// TwinCAT 3 PLC project System
// ProgramVersion: 3.1.4023.0
// libraries:
//   Tc2_MC2, * (Beckhoff Automation GmbH)
//   Tc2_MC2_Drive, * (Beckhoff Automation GmbH)
//   Tc2_Standard, * (Beckhoff Automation GmbH)
//   Tc2_System, * (Beckhoff Automation GmbH)
//   Tc3_Module, * (Beckhoff Automation GmbH)
// project tree:
//   00_Internal PackAL/DUTs/ E_PMLState.TcDUT (not stored), E_PMLUnitMode.TcDUT
//   00_Internal PackAL/POUs/ PS_PackML_StateMachine_Auto.TcPOU, PS_PackML_StateMachine_Maintenance.TcPOU, PS_PackML_StateMachine_Manual.TcPOU, PS_PackML_StateMachine_SemiAuto.TcPOU, PS_UnitModeManager.TcPOU
//   01_Submodules/ FB_Axis.TcPOU, FB_MPG.TcPOU
//   02_Subsystems/ FB_Stage.TcPOU
//   03_Machine/ FB_Machine.TcPOU
//   04_Application/ MAIN.TcPOU
//   05_Visu/ FB_Visu.TcPOU, HMI.TcVIS, TAB_Simulation.TcVIS
//   DUTs/ ST_MC_Base.TcDUT, ST_MC_CMD.TcDUT, ST_MC_Reset.TcDUT, ST_MC_Status.TcDUT
//   / GlobalTextList.TcGTLO, PlcTask.TcTTO, Visualization Manager.TcVMO (not stored), VISU_TASK.TcTTO
//   GVLs/ GVL_SA.TcGVL, Temp.TcGVL
//   POUs/ FB_MotorControl.TcPOU, ModbusTCP_Test.TcPOU
// real-time tasks:
//   TASK PlcTask: cycle T#10ms, priority 20, ADS port 350
//   TASK VISU_TASK: cycle T#100000us, priority 30, ADS port 351
// motion (NC):
//   TASK NC-Task 1 SAF: cycle T#2ms, priority 4, ADS port 501
//   TASK NC-Task 1 SVB: cycle T#10ms, priority 8, ADS port 511
//   AXIS Axis 2 (id 2)
//     OtherSettings: AllowMotionCmdToSlave=true
//     encoder EncType=19
//       EncPara: MaxCount=#xffffffff
//     drive DrvType=16
//       DrvPara: MaxCount=#xffffffff, DriveControlDWord=#x00020000
//         Analog: TorqueSetpointScale=10, ScaleFactorActTorque=0.1
//         TimeComp: TaskDelayCycles=1
//     controller CtrType=1
//       CtrPara: PriorControlFactor=1
//         Observer: BandWidth=20
// I/O:
//   DEVICE Device 3 (EtherCAT), AmsNetId 129.169.49.186.4.1
//     Term 1 (EK1100) [EK1100 EtherCAT Coupler (2A E-Bus)] (disabled)
//       Term 2 (EL1114)
//       Term 3 (EL1809) [EL1809 16Ch. Dig. Input 24V, 3ms]
//       Term 4 (EL1809) [EL1809 16Ch. Dig. Input 24V, 3ms]
//       Term 5 (EL2008) [EL2008 8Ch. Dig. Output 24V, 0.5A]
//       Term 6 (EL2809) [EL2809 16Ch. Dig. Output 24V, 0.5A]
//       Term 7 (EL3068) [EL3068 8Ch. Ana. Input 0-10V]
//       Term 8 (EL3058) [EL3058 8Ch. Ana. Input 4-20mA]
//       Term 9 (EL4002) [EL4002 2Ch. Ana. Output 0-10V, 12bit]
//       Term 10 (EL5101) [EL5101 1Ch. Inc. Encoder 5V]
//       Term 11 (EK1110) [EK1110 EtherCAT extension]
//   DEVICE Device 1 (EtherCAT) (disabled), AmsNetId 192.168.1.163.2.1
//     Term 1 (EK1200) [EK1200-5000 EtherCAT Power supply (2A E-Bus)]
//       Term 13 (EL1114) [EL1114 4Ch. Dig. Input 24V, 10µs, Sensor Power]
//       Term 14 (EL1809) [EL1809 16Ch. Dig. Input 24V, 3ms]
//       Term 15 (EL1809) [EL1809 16Ch. Dig. Input 24V, 3ms]
//       Term 16 (EL2008) [EL2008 8Ch. Dig. Output 24V, 0.5A]
//       Term 17 (EL2809) [EL2809 16Ch. Dig. Output 24V, 0.5A]
//       Term 18 (EL3068) [EL3068 8Ch. Ana. Input 0-10V]
//       Term 19 (EL3058) [EL3058 8Ch. Ana. Input 4-20mA]
//       Term 20 (EL4002) [EL4002 2Ch. Ana. Output 0-10V, 12bit]
//       Term 21 (EL5101) [EL5101 1Ch. Inc. Encoder 5V]
//       Term 22 (EK1110) [EK1110 EtherCAT extension]
//   DEVICE Device 5 (NOV-DP-RAM)
// variable links:
//   System Instance <-> Device 3 (EtherCAT)/Term 1 (EK1100)/Term 10 (EL5101)
//     PlcTask Inputs/MAIN.fbMachine.fbMPG.EncoderValue <-> ENC Status compact/Counter value
//   System Instance <-> NC-Task 1 SAF/Axes/Axis 2
//     PlcTask Inputs/GVL_SA.Motor1.AxisRef.NcToPlc <-> Outputs/ToPlc
//     PlcTask Outputs/GVL_SA.Motor1.AxisRef.PlcToNc <-> Inputs/FromPlc

CONFIGURATION System
    RESOURCE PLC ON TwinCAT3
        TASK PlcTask(INTERVAL := T#10ms, PRIORITY := 20);
        TASK VISU_TASK(INTERVAL := T#100000us, PRIORITY := 30);
        PROGRAM MAIN WITH PlcTask : MAIN;
        PROGRAM VisuElems_Visu_Prg WITH VISU_TASK : VisuElems.Visu_Prg;
    END_RESOURCE
END_CONFIGURATION

// ---- 00_Internal PackAL/DUTs/E_PMLUnitMode.TcDUT
{attribute 'qualified_only'}
{attribute 'strict'}
TYPE E_PMLUnitMode :
(
	UNDEFINED		:=  0,
	AUTOMATIC		:=  1,
	MAINTENANCE 	:=  2,
	MANUAL 			:=  3,
	SEMIAUTOMATIC	:=  4,
	DRYRUN			:=  5,
	USERMODE1		:=  6,
	USERMODE2		:=  7,
	IDLE 			:=  8,
	ESTOP 			:=  9
);
END_TYPE

// ---- DUTs/ST_MC_Base.TcDUT
TYPE ST_MC_Base :
STRUCT
	Busy		:	BOOL;
	Error		:	BOOL;
	ErrrorID	:	UDINT;
END_STRUCT
END_TYPE

// ---- DUTs/ST_MC_CMD.TcDUT
TYPE ST_MC_CMD :
STRUCT
	bExe			: BOOL	;
	lrVelocity		: LREAL	;
	lrAcceleration 	: LREAL ;
	lrDeceleration 	: LREAL ;
	lrJerk 			: LREAL ;
	lrDistance 		: LREAL ; 
	lrPosition 		: LREAL ; 
	EnuDirection 	: MC_Direction ;
	EnuBufferMode 	: MC_BufferMode ; 
	EnuOptions 		: ST_MoveOptions ;
END_STRUCT
END_TYPE

// ---- DUTs/ST_MC_Reset.TcDUT
TYPE ST_MC_Reset:
STRUCT
	
	CMD_Execute	: 	BOOL;
	
	Done		: 	BOOL;
	Busy		:	BOOL;
	Error		:	BOOL;
	ErrrorID	:	UDINT;	

END_STRUCT
END_TYPE

// ---- DUTs/ST_MC_Status.TcDUT
TYPE ST_MC_Status :
STRUCT
	
	Status		:	BOOL;
	Done		:	BOOL;
	Busy		:	BOOL;
	Error		:	BOOL;
	Active		:	BOOL;
	CmdAborted	:	BOOL;
	InVelocity	:	BOOL;
	ErrrorID	:	UDINT;
	
	Value		: 	LREAL;
	Valid		: 	BOOL;
	

END_STRUCT
END_TYPE

// ---- GVLs/GVL_SA.TcGVL
{attribute 'qualified_only'}
VAR_GLOBAL
	Motor1 : FB_MotorControl;	
END_VAR

// ---- GVLs/Temp.TcGVL
{attribute 'qualified_only'}
VAR_GLOBAL
	//GVL_MPG_Value : UINT;
	
	bSwitch1:	BOOL;
	bLED1: BOOL;
	
	
END_VAR

// ---- 04_Application/MAIN.TcPOU
PROGRAM MAIN
VAR
	fbMachine : FB_Machine;	

	Dummy : BOOL := FALSE;
	bTest: BOOL := FALSE;
	
	MAIN_UINT : UINT;
	
END_VAR

// =========================================================

fbMachine();

// =========================================================


//GVL_SA.Motor1.UpdateAll();
GVL_SA.Motor1();

GVL_SA.Motor1.bStateEnable := TRUE;

{IF defined (Pyrometer_Motor)}
	bTest := TRUE;
{END_IF}

Dummy	:= TRUE;

Temp.bLED1 := Temp.bSwitch1;

END_PROGRAM

// ---- 03_Machine/FB_Machine.TcPOU
FUNCTION_BLOCK FB_Machine
VAR_INPUT
	
END_VAR
VAR_OUTPUT
END_VAR
VAR
	// =============== Common variables =========================================================
	bInit								: BOOL;									// True if module parameters are initialized	

		
	
	// =============== Machine elements =========================================================
	// This can be either Submodules or SubSystems
	fbMPG 			: 		FB_MPG ;		//MPG unit
	
	
	
	fbVisu : FB_Visu;
	
		fbGetCurTaskIndex : GETCURTASKINDEX;
	
	// =============== Testing ==================================================================
	_UINT : UINT;
END_VAR

// =========================================================
// Call of actions

//Check for start cycle
//Move to main later.....
//fbGetCurTaskIndex();
//IF _TaskInfo[fbGetCurTaskIndex.index].FirstCycle THEN
//    // The code that you want to be executed at the first cycle
//	eMPGState := INIT_START;
//END_IF


	// Init
	General_Init();

	// Mode and state requests
	//General_Requests();
	
	// Enable for power supply, compressed air control and buttons
	//General_Enable();
	
	// Input variables of separating and sorting modules
	//General_ModuleInputs();
	
	// Output variables
	//General_SetOutput();
	
	// State machine
	//General_StateMachine();
	
	// Visualization
	//General_Visu();
	fbVisu();
	

// =========================================================
//TESTING


	_UINT := fbMPG.Value;

METHOD PRIVATE General_Init
VAR_INPUT
		
END_VAR
// =========================================================
IF NOT bInit THEN
		fbMPG.Start(1234);
		
	// Init done
		bInit := TRUE;
END_IF
// =========================================================
END_METHOD

METHOD PRIVATE Operating_Automatic
VAR_INPUT
END_VAR
END_METHOD

METHOD PRIVATE Operating_Manual
VAR_INPUT
END_VAR
END_METHOD

END_FUNCTION_BLOCK

// ---- 01_Submodules/FB_MPG.TcPOU
FUNCTION_BLOCK FB_MPG
VAR_INPUT
END_VAR
VAR_OUTPUT
END_VAR
VAR
	//Hardware declared here as only one will ever be connected 
	EncoderValue 		AT %I* : UINT;	//Measured Value from Encoder
	SetValueZero	 	AT %Q* : BOOL;	//Request encoder be reset to zero 	
	bX1					AT %I* : BOOL;	//Multipliers
	bX10				AT %I* : BOOL;
	bX100				AT %I* : BOOL;
	bEnabled			AT %I* : BOOL;
	
	
	eMPGState : (INIT_START, WAIT_START, RUNNING, STOPPED);	//MPG state machine defenitions
	
	nMotorStartPoisition	: UINT	;	//Where was the motor at the beginning
	nDeltaPosition			: DINT	;	//Calculated position request change from start
										//Motor value 	nMotorStartPoisition + nDeltaPosition

	nLastEncoderValue		: UINT	;	//Encoder value on last scan cycle
	nDeltaEncoder_PerScan	: DINT	;	//Encoder change per scan
	
END_VAR

CASE eMPGState OF
	INIT_START:												//Holding state
		eMPGState := WAIT_START;
	
	WAIT_START:												//Holding state
		eMPGState := RUNNING;

	RUNNING:
		IF (Error_Scaler OR Error_AxisSelect) THEN			//If current error state
			//nDeltaPosition := 0;							//No change in position possible	
		ELSE
			//Update values
			nDeltaEncoder_PerScan  := nLastEncoderValue - EncoderValue;
			nDeltaPosition := nDeltaPosition + nDeltaEncoder_PerScan * ScaleFactor;			
		END_IF

	STOPPED:
		//Do nothing
END_CASE

nLastEncoderValue := EncoderValue;	//Ensure next scan always sees change in encoder position

PROPERTY PUBLIC Error : Bool
GET
//System in any error or any condition other than running.

Error := FALSE;

IF (Error_AxisSelect OR Error_Scaler) THEN
	Error := TRUE;
END_IF

IF eMPGState <> RUNNING THEN
	Error := TRUE;
END_IF
END_GET
END_PROPERTY

PROPERTY PRIVATE Error_AxisSelect : Bool
GET
END_GET
END_PROPERTY

PROPERTY PRIVATE Error_Scaler : Bool
GET
//Error conditions
IF bX1 AND bX10 THEN
	Error_Scaler := TRUE;
	RETURN;
END_IF

IF bX1 AND bX100 THEN
	Error_Scaler := TRUE;
	RETURN;
END_IF

IF bX10 AND bX100 THEN
	Error_Scaler := TRUE;
	RETURN;
END_IF

IF NOT bX1 AND NOT bX10 AND NOT bX100 THEN
	Error_Scaler := TRUE;
	RETURN;
END_IF

Error_Scaler := FALSE;
END_GET
END_PROPERTY

//Returns the scale factor to be used on the new data
PROPERTY PRIVATE ScaleFactor : UINT
GET
//Depending on what IO is connected send back 1, 10, 100 or set error!
IF bX1 THEN
	ScaleFactor := 1;
END_IF

IF bX10 THEN
	ScaleFactor := 10;
END_IF

IF bX100 THEN
	ScaleFactor := 100;
END_IF
END_GET
END_PROPERTY

METHOD PUBLIC Start
VAR_INPUT
	nMotorStartPoisition	:	UINT ;	//Check that this is passed to the "main"
										//May need to be implicitly defined.
END_VAR
eMPGState := INIT_START;
END_METHOD

PROPERTY Starting : Bool
GET
IF (eMPGState = INIT_START OR eMPGState = WAIT_START) THEN
	Starting := TRUE;
	ELSE
	Starting := FALSE;				
END_IF
END_GET
END_PROPERTY

METHOD PUBLIC Stop
VAR_INPUT
END_VAR
eMPGState := E_PMLState.STOPPED;
END_METHOD

PROPERTY Value : UINT		//Calculated ABS position value requested by MPG, check Error before use.
GET
Value := DINT_TO_UINT(nMotorStartPoisition + nDeltaPosition);
//What is the form needed for motor position??
END_GET
END_PROPERTY

END_FUNCTION_BLOCK

// ---- 05_Visu/FB_Visu.TcPOU
FUNCTION_BLOCK FB_Visu
VAR_INPUT
	nMPGCounter : DINT;
END_VAR
VAR_OUTPUT
END_VAR
VAR
	sDisplayText_MPG : STRING(15);
END_VAR

sDisplayText_MPG := 'Sent';

END_FUNCTION_BLOCK

// ---- POUs/FB_MotorControl.TcPOU
FUNCTION_BLOCK FB_MotorControl
VAR_INPUT
	AxisRef 	:	AXIS_REF;
	//Position
	//Ready
	//Reset
	
END_VAR
VAR_OUTPUT
		error	: BOOL;
END_VAR

(*Internals*)
VAR
	(* Properties *)
	Enabled : BOOL := FALSE;	


	eInitMotor : (START, IN_PROCESS, DONE, ERROR);	
	eMoveABS : (START, IN_PROCESS, DONE, ERROR);

	//stMC_Reset : ST_MC_Reset;
	

	stSA_Reset	:   ST_MC_Status;
	
	
	
	fbMcPower	:	MC_POWER;
	fbMcHome	: 	MC_HOME;
	fbMcJog		:	MC_JOG;
	
	// Global
	bError 		: BOOL	; // := TRUE;
	nErrorID 	: LINT	; //Check type
	
	//Reset
	fbMcReset	:	MC_RESET;
	fbTriggerReset : R_TRIG;
	bResetDone : BOOL := FALSE;
	
	
	
	fbMoveVelocity	: MC_MoveVelocity;
	fbMoveRelative	: MC_MoveRelative;
	fbMoveAbsolute	: MC_MoveAbsolute;
	
	fbHalt	: MC_Halt;
	fbStop	: MC_Stop;
	
	fbSA_GetPosition : MC_ReadActualPosition;
	
	//Input: Command
	bCmdResetExe			:	BOOL	;
	bCmdPowerEnable			:	BOOL	;
	bCmdPowerEnablePositive	:	BOOL	;
	bCmdPowerEnableNegative	:	BOOL	;
	bCmdHomeExecute			:	BOOL	;
	bSA_HomeCamInput	:	BOOL	;
	
	bSA_JogFwd			:	BOOL	;
	bSA_JogRev			:	BOOL	;
	
	bSA_HaltExe			: 	BOOL	;
	bSA_StopExe			: 	BOOL	;
	
	//stStatusMoveVelocity	: ST_MC_CMD	;
	stSA_VelCmd1	: ST_MC_CMD;
	stSA_RelCmd1			: ST_MC_CMD	;
	stSA_AbsCmd1			: ST_MC_CMD	;
	
	//Variables / Parameters
	lrSA_PowerOverride	: LREAL;
	lrSA_HomePosition	: LREAL;
	lrSA_SetPosition	: LREAL;
	lrSA_JogVelocity	: LREAL;
	
	//Status
	//stSA_Reset			: ST_MC_Status;
	stSA_Power			: ST_MC_Status;
	stSA_Home			: ST_MC_Status;
	stSA_SetPosition	: ST_MC_Status;
	stSA_Jog			: ST_MC_Status;
	stSA_GetPosition	: ST_MC_Status;
	
	
	stSA_VelSts1		: ST_MC_Status;
	stSA_MoveRelative		: ST_MC_Status;
	stSA_AbsSts1		: ST_MC_Status;
	
	stSA_Halt			: ST_MC_Status;
	stSA_Stop			: ST_MC_Status;

END_VAR

AxisRef.ReadStatus();
GetStatus();
//Here the state machine needs to be processed or farmed out.



//For a move

//Has position changed from the current target.....






//This should be removed as seperate methods are added.
ExecuteCommands();

PROPERTY bStateEnable : BOOL
GET
bStateEnable := Enabled ;
END_GET
SET
Enabled := bStateEnable;
END_SET
END_PROPERTY

METHOD PRIVATE Enable : BOOL
VAR_INPUT
END_VAR
END_METHOD

METHOD PRIVATE ExecuteCommands : BOOL
VAR_INPUT
END_VAR

VAR
END_VAR
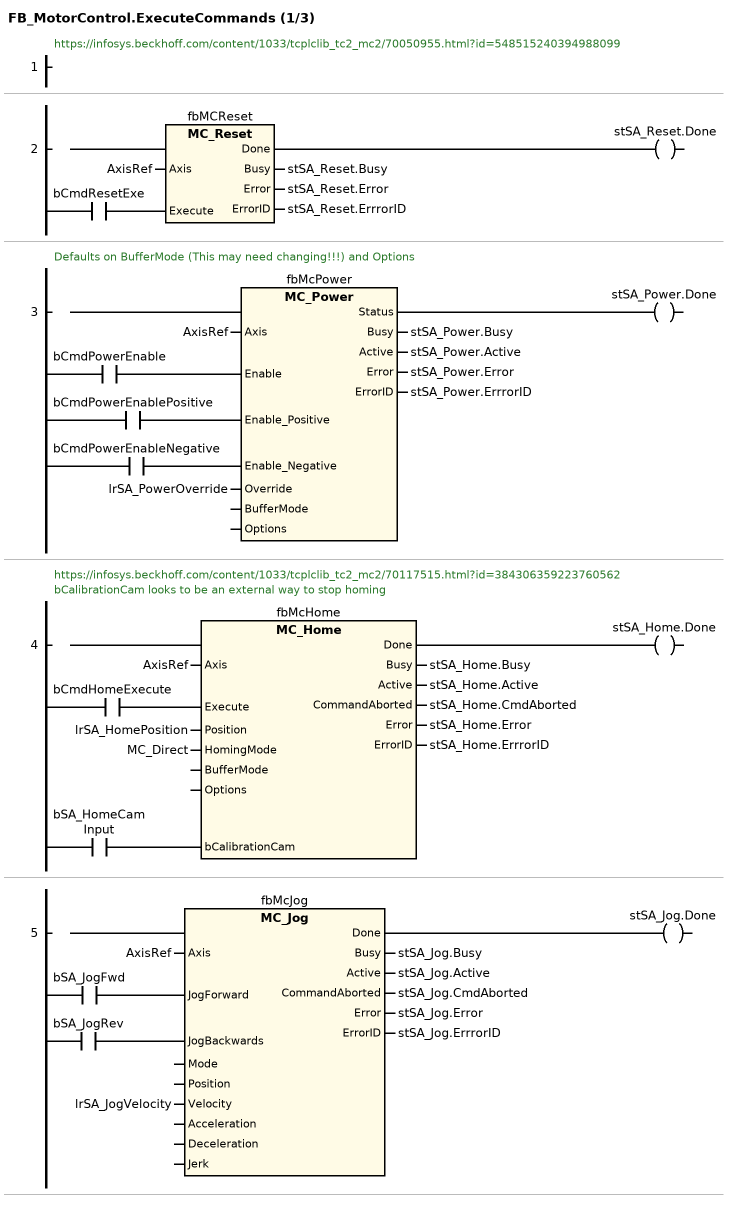
// NETWORK 1
// https://infosys.beckhoff.com/content/1033/tcplclib_tc2_mc2/70050955.html?id=548515240394988099

// NETWORK 2
fbMCReset(
    Axis := AxisRef,
    Execute := bCmdResetExe,
    Busy => stSA_Reset.Busy,
    Error => stSA_Reset.Error,
    ErrorID => stSA_Reset.ErrrorID); // MC_Reset
stSA_Reset.Done := fbMCReset.Done;

// NETWORK 3
// Defaults on BufferMode (This may need changing!!!) and Options
fbMcPower(
    Axis := AxisRef,
    Enable := bCmdPowerEnable,
    Enable_Positive := bCmdPowerEnablePositive,
    Enable_Negative := bCmdPowerEnableNegative,
    Override := lrSA_PowerOverride,
    Busy => stSA_Power.Busy,
    Active => stSA_Power.Active,
    Error => stSA_Power.Error,
    ErrorID => stSA_Power.ErrrorID); // MC_Power
stSA_Power.Done := fbMcPower.Status;

// NETWORK 4
// https://infosys.beckhoff.com/content/1033/tcplclib_tc2_mc2/70117515.html?id=384306359223760562
// bCalibrationCam looks to be an external way to stop homing
fbMcHome(
    Axis := AxisRef,
    Execute := bCmdHomeExecute,
    Position := lrSA_HomePosition,
    HomingMode := MC_Direct,
    bCalibrationCam := bSA_HomeCamInput,
    Busy => stSA_Home.Busy,
    Active => stSA_Home.Active,
    CommandAborted => stSA_Home.CmdAborted,
    Error => stSA_Home.Error,
    ErrorID => stSA_Home.ErrrorID); // MC_Home
stSA_Home.Done := fbMcHome.Done;

// NETWORK 5
fbMcJog(
    Axis := AxisRef,
    JogForward := bSA_JogFwd,
    JogBackwards := bSA_JogRev,
    Velocity := lrSA_JogVelocity,
    Busy => stSA_Jog.Busy,
    Active => stSA_Jog.Active,
    CommandAborted => stSA_Jog.CmdAborted,
    Error => stSA_Jog.Error,
    ErrorID => stSA_Jog.ErrrorID); // MC_Jog
stSA_Jog.Done := fbMcJog.Done;

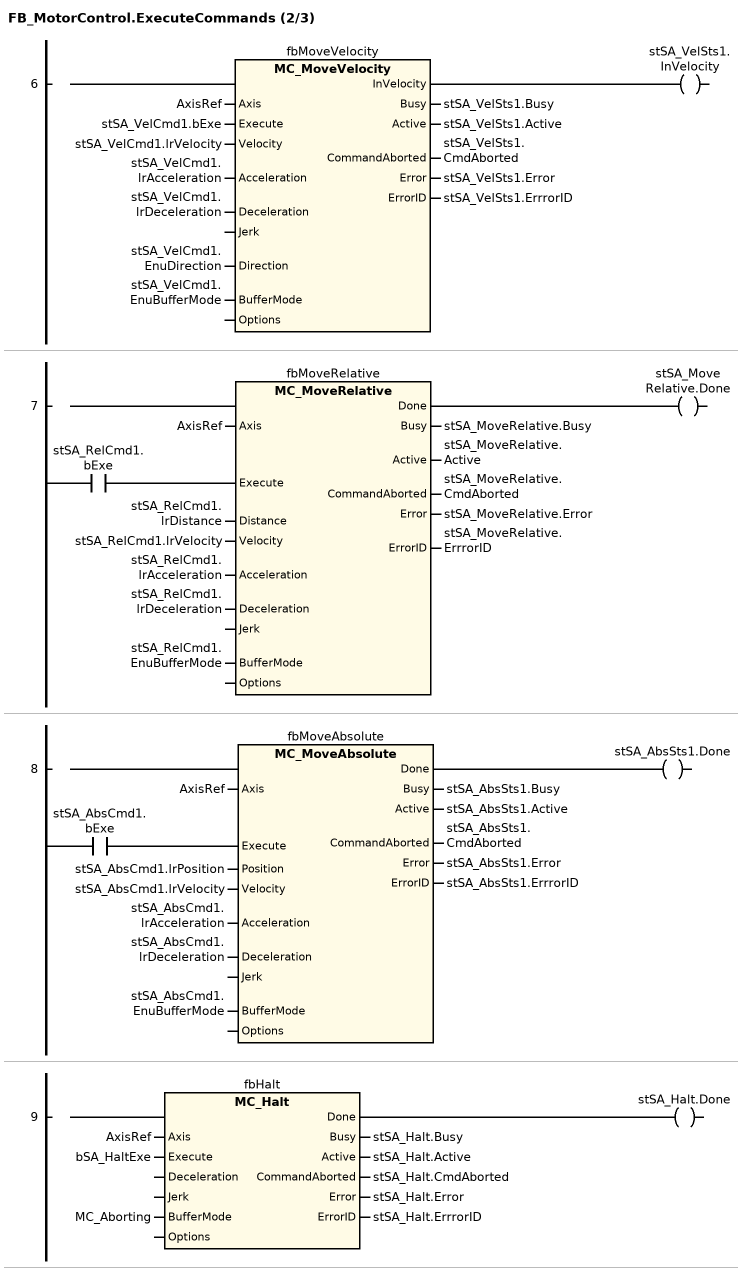
// NETWORK 6
fbMoveVelocity(
    Axis := AxisRef,
    Execute := stSA_VelCmd1.bExe,
    Velocity := stSA_VelCmd1.lrVelocity,
    Acceleration := stSA_VelCmd1.lrAcceleration,
    Deceleration := stSA_VelCmd1.lrDeceleration,
    Direction := stSA_VelCmd1.EnuDirection,
    BufferMode := stSA_VelCmd1.EnuBufferMode,
    Busy => stSA_VelSts1.Busy,
    Active => stSA_VelSts1.Active,
    CommandAborted => stSA_VelSts1.CmdAborted,
    Error => stSA_VelSts1.Error,
    ErrorID => stSA_VelSts1.ErrrorID); // MC_MoveVelocity
stSA_VelSts1.InVelocity := fbMoveVelocity.InVelocity;

// NETWORK 7
fbMoveRelative(
    Axis := AxisRef,
    Execute := stSA_RelCmd1.bExe,
    Distance := stSA_RelCmd1.lrDistance,
    Velocity := stSA_RelCmd1.lrVelocity,
    Acceleration := stSA_RelCmd1.lrAcceleration,
    Deceleration := stSA_RelCmd1.lrDeceleration,
    BufferMode := stSA_RelCmd1.EnuBufferMode,
    Busy => stSA_MoveRelative.Busy,
    Active => stSA_MoveRelative.Active,
    CommandAborted => stSA_MoveRelative.CmdAborted,
    Error => stSA_MoveRelative.Error,
    ErrorID => stSA_MoveRelative.ErrrorID); // MC_MoveRelative
stSA_MoveRelative.Done := fbMoveRelative.Done;

// NETWORK 8
fbMoveAbsolute(
    Axis := AxisRef,
    Execute := stSA_AbsCmd1.bExe,
    Position := stSA_AbsCmd1.lrPosition,
    Velocity := stSA_AbsCmd1.lrVelocity,
    Acceleration := stSA_AbsCmd1.lrAcceleration,
    Deceleration := stSA_AbsCmd1.lrDeceleration,
    BufferMode := stSA_AbsCmd1.EnuBufferMode,
    Busy => stSA_AbsSts1.Busy,
    Active => stSA_AbsSts1.Active,
    CommandAborted => stSA_AbsSts1.CmdAborted,
    Error => stSA_AbsSts1.Error,
    ErrorID => stSA_AbsSts1.ErrrorID); // MC_MoveAbsolute
stSA_AbsSts1.Done := fbMoveAbsolute.Done;

// NETWORK 9
fbHalt(
    Axis := AxisRef,
    Execute := bSA_HaltExe,
    BufferMode := MC_Aborting,
    Busy => stSA_Halt.Busy,
    Active => stSA_Halt.Active,
    CommandAborted => stSA_Halt.CmdAborted,
    Error => stSA_Halt.Error,
    ErrorID => stSA_Halt.ErrrorID); // MC_Halt
stSA_Halt.Done := fbHalt.Done;

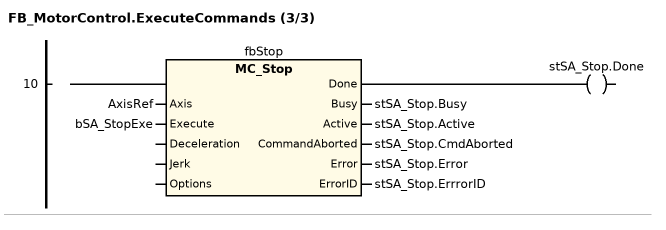
// NETWORK 10
fbStop(
    Axis := AxisRef,
    Execute := bSA_StopExe,
    Busy => stSA_Stop.Busy,
    Active => stSA_Stop.Active,
    CommandAborted => stSA_Stop.CmdAborted,
    Error => stSA_Stop.Error,
    ErrorID => stSA_Stop.ErrrorID); // MC_Stop
stSA_Stop.Done := fbStop.Done;
END_METHOD

METHOD PRIVATE GetStatus : BOOL
VAR_INPUT
END_VAR
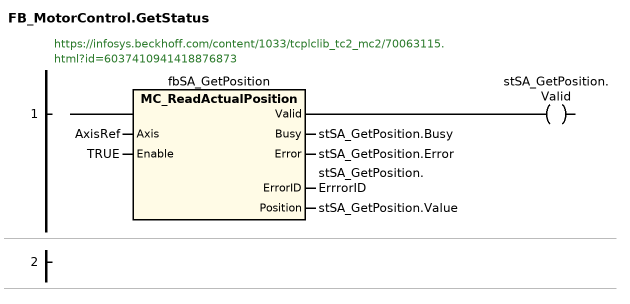
// NETWORK 1
// https://infosys.beckhoff.com/content/1033/tcplclib_tc2_mc2/70063115.html?id=6037410941418876873
fbSA_GetPosition(
    Axis := AxisRef,
    Enable := TRUE,
    Busy => stSA_GetPosition.Busy,
    Error => stSA_GetPosition.Error,
    ErrorID => stSA_GetPosition.ErrrorID,
    Position => stSA_GetPosition.Value); // MC_ReadActualPosition
stSA_GetPosition.Valid := fbSA_GetPosition.Valid;

// NETWORK 2
END_METHOD

METHOD Halt : BOOL
VAR_INPUT
END_VAR
END_METHOD

METHOD PUBLIC MoveAbs : BOOL
VAR_INPUT
	Distance 		: LREAL;
	Velocity 		: LREAL;

//https://infosys.beckhoff.com/content/1033/tcplclib_tc2_mc2/70147595.html?id=4401319670753010232
	mcBufferMode	: MC_BufferMode;
(*  MC_Aborting,			Cancels P1 and  moves to P2
    MC_Buffered,			Moves to P1, stops and moves to P2
    MC_BlendingLow, MC_BlendingPrevious, MC_BlendingNext, MC_BlendingHigh	Change the way speed is blended  BlendingLow would generaly be the one I'd choose. *)
	
END_VAR
VAR
	

END_VAR
(*  It is not needed to wait for the end of a move, will be qued - but do need to ensure Execute operates with a rising edge.
	Not concerned about "loosing" commands, no buffer needed, only the last command matters.*)   

(*
If in Error state ignore.

If "Busy"	Execute == FALSE;

if Execute == FALSE can send new command

*)	

	
	
//CASE fbMoveAbsolute.Execute OF
//	TRUE: 
	
//	IN_PROCESS:

//	DONE:
	
	
//END_CASE

//Does this have meaning.....
MoveAbs := TRUE;
END_METHOD

METHOD Reset : BOOL
VAR_INPUT
	bDriveReset : Bool;
END_VAR
// Indicate that the Reset is in progress
IF NOT bDriveReset THEN
	bResetDone := FALSE;
END_IF

// Trigger
fbTriggerReset(CLK := bDriveReset);

IF fbTriggerReset.Q THEN
	//Is this meant to be sending a halt to the motor at the same time....?
	//If so why not as a command - seems more of a status....
	
	//bHaltDone := FALSE;
	fbMcReset(Execute := TRUE, Axis := AxisRef);
ELSE				
	fbMcReset(Axis := AxisRef); //What happens to the unchanged values - defaults......TEST?
END_IF;
 
// Done / Error 
IF fbMcReset.Done OR fbMcReset.Error THEN
	bError := fbMcReset.Error;
	nErrorID := fbMcReset.ErrorID;
	bResetDone := fbMcReset.Done;
	
	fbMcReset(Execute := FALSE, Axis := AxisRef);
END_IF
END_METHOD

METHOD Stop : BOOL
VAR_INPUT
END_VAR
END_METHOD

END_FUNCTION_BLOCK

// ---- 00_Internal PackAL/POUs/PS_PackML_StateMachine_Auto.TcPOU
FUNCTION_BLOCK PS_PackML_StateMachine_Auto
VAR_INPUT
	Start				: BOOL;
	Hold				: BOOL;
	UnHold				: BOOL;
	Suspend				: BOOL;
	UnSuspend			: BOOL;
	Abort				: BOOL;
	Stop				: BOOL;
	Complete			: BOOL;
	Clear				: BOOL;
	Reset				: BOOL;
	StateComplete		: BOOL;
END_VAR
VAR_OUTPUT
	Status				: WORD;

	ST_Starting			: BOOL;
	ST_Completing		: BOOL;
	ST_Resetting		: BOOL;
	ST_Holding			: BOOL;
	ST_UnHolding		: BOOL;
	ST_Suspending		: BOOL;
	ST_UnSuspending		: BOOL;
	ST_Clearing			: BOOL;
	ST_Stopping			: BOOL;
	ST_Aborting			: BOOL;

	(* State Complete*)
	ST_Execute			: BOOL;
	ST_Complete			: BOOL;
	ST_Idle				: BOOL;
	ST_Held				: BOOL;
	ST_Suspended		: BOOL;
	ST_Stopped			: BOOL;
	ST_Aborted			: BOOL;

	(* additional *)
	Error				: BOOL;
	ErrorID				: DWORD;
	ePMLState			: E_PMLState := E_PMLState.IDLE;
END_VAR
VAR
	ePMLStatePrev		: E_PMLState;
	bStateChange		: BOOL;
	StateCompletePrev	: BOOL;
END_VAR

(* check for state change *)
IF ePMLStatePrev <> ePMLState THEN
	ePMLStatePrev 	:= ePMLState;
	bStateChange	:= TRUE;
ELSE
	bStateChange	:= FALSE;
END_IF


(* change to new state if requested *)
CASE ePMLState OF
	E_PMLState.UNDEFINED:
				(* undefined state *)
				IF bStateChange THEN
					(* transient state *)
					ST_Starting		:= FALSE;
					ST_Completing	:= FALSE;
					ST_Resetting	:= FALSE;
					ST_Holding		:= FALSE;
					ST_UnHolding	:= FALSE;
					ST_Suspending	:= FALSE;
					ST_UnSuspending	:= FALSE;
					ST_Clearing		:= FALSE;
					ST_Stopping		:= FALSE;
					ST_Aborting		:= FALSE;
		
					(* final state *)
					ST_Execute		:= FALSE;
					ST_Complete		:= FALSE;
					ST_Idle			:= FALSE;
					ST_Held			:= FALSE;
					ST_Suspended	:= FALSE;
					ST_Stopped		:= FALSE;
					ST_Aborted		:= FALSE;
				END_IF
		
				IF Abort THEN
					ePMLState 		:= E_PMLState.ABORTING;
					ST_Aborting		:= TRUE;
				ELSIF Stop THEN
					ePMLState 		:= E_PMLState.STOPPING;
					ST_Stopping		:= TRUE;
				END_IF


	E_PMLState.IDLE:
				(* final state *)
		
				IF bStateChange THEN
					(* transient state *)
					ST_Starting		:= FALSE;
					ST_Completing	:= FALSE;
					ST_Resetting	:= FALSE;
					ST_Holding		:= FALSE;
					ST_UnHolding	:= FALSE;
					ST_Suspending	:= FALSE;
					ST_UnSuspending	:= FALSE;
					ST_Clearing		:= FALSE;
					ST_Stopping		:= FALSE;
					ST_Aborting		:= FALSE;
		
					(* final state *)
					ST_Execute		:= FALSE;
					ST_Complete		:= FALSE;
					ST_Idle			:= TRUE;
					ST_Held			:= FALSE;
					ST_Suspended	:= FALSE;
					ST_Stopped		:= FALSE;
					ST_Aborted		:= FALSE;
				END_IF
		
				IF Abort THEN
					ePMLState 		:= E_PMLState.ABORTING;
					ST_Idle			:= FALSE;
					ST_Aborting		:= TRUE;
				ELSIF Stop THEN
					ePMLState 		:= E_PMLState.STOPPING;
					ST_Idle			:= FALSE;
					ST_Stopping		:= TRUE;
				ELSIF Start THEN
					ePMLState 		:= E_PMLState.STARTING;
					ST_Idle			:= FALSE;
					ST_Starting		:= TRUE;
				END_IF


	E_PMLState.STARTING:
				(* transient state *)
		
				IF bStateChange THEN
					(* transient state *)
					ST_Starting		:= TRUE;
					ST_Completing	:= FALSE;
					ST_Resetting	:= FALSE;
					ST_Holding		:= FALSE;
					ST_UnHolding	:= FALSE;
					ST_Suspending	:= FALSE;
					ST_UnSuspending	:= FALSE;
					ST_Clearing		:= FALSE;
					ST_Stopping		:= FALSE;
					ST_Aborting		:= FALSE;
		
					(* final state *)
					ST_Execute		:= FALSE;
					ST_Complete		:= FALSE;
					ST_Idle			:= FALSE;
					ST_Held			:= FALSE;
					ST_Suspended	:= FALSE;
					ST_Stopped		:= FALSE;
					ST_Aborted		:= FALSE;
				END_IF
		
				IF Abort THEN
					ePMLState 		:= E_PMLState.ABORTING;
					ST_Starting		:= FALSE;
					ST_Aborting		:= TRUE;
				ELSIF Stop THEN
					ePMLState 		:= E_PMLState.STOPPING;
					ST_Starting		:= FALSE;
					ST_Stopping		:= TRUE;
				ELSIF StateComplete AND NOT StateCompletePrev THEN
					ePMLState 		:= E_PMLState.EXECUTE;
					StateCompletePrev := StateComplete;
					ST_Starting		:= FALSE;
					ST_Execute		:= TRUE;
				END_IF


	E_PMLState.EXECUTE:
				(* final state *)
		
				IF bStateChange THEN
					(* transient state *)
					ST_Starting		:= FALSE;
					ST_Completing	:= FALSE;
					ST_Resetting	:= FALSE;
					ST_Holding		:= FALSE;
					ST_UnHolding	:= FALSE;
					ST_Suspending	:= FALSE;
					ST_UnSuspending	:= FALSE;
					ST_Clearing		:= FALSE;
					ST_Stopping		:= FALSE;
					ST_Aborting		:= FALSE;
		
					(* final state *)
					ST_Execute		:= TRUE;
					ST_Complete		:= FALSE;
					ST_Idle			:= FALSE;
					ST_Held			:= FALSE;
					ST_Suspended	:= FALSE;
					ST_Stopped		:= FALSE;
					ST_Aborted		:= FALSE;
				END_IF
		
				IF Abort THEN
					ePMLState 		:= E_PMLState.ABORTING;
					ST_Execute		:= FALSE;
					ST_Aborting		:= TRUE;
				ELSIF Stop THEN
					ePMLState 		:= E_PMLState.STOPPING;
					ST_Execute		:= FALSE;
					ST_Stopping		:= TRUE;
				ELSIF Suspend THEN
					ePMLState 		:= E_PMLState.SUSPENDING;
					ST_Execute		:= FALSE;
					ST_Suspending	:= TRUE;
				ELSIF Hold THEN
					ePMLState 		:= E_PMLState.HOLDING;
					ST_Execute		:= FALSE;
					ST_Holding		:= TRUE;
				ELSIF Complete THEN
					ePMLState 		:= E_PMLState.COMPLETING;
					ST_Execute		:= FALSE;
					ST_Completing	:= TRUE;
				END_IF


	E_PMLState.COMPLETING:
				(* transient state *)
		
				IF bStateChange THEN
					(* transient state *)
					ST_Starting		:= FALSE;
					ST_Completing	:= TRUE;
					ST_Resetting	:= FALSE;
					ST_Holding		:= FALSE;
					ST_UnHolding	:= FALSE;
					ST_Suspending	:= FALSE;
					ST_UnSuspending	:= FALSE;
					ST_Clearing		:= FALSE;
					ST_Stopping		:= FALSE;
					ST_Aborting		:= FALSE;
		
					(* final state *)
					ST_Execute		:= FALSE;
					ST_Complete		:= FALSE;
					ST_Idle			:= FALSE;
					ST_Held			:= FALSE;
					ST_Suspended	:= FALSE;
					ST_Stopped		:= FALSE;
					ST_Aborted		:= FALSE;
				END_IF
		
				IF Abort THEN
					ePMLState 		:= E_PMLState.ABORTING;
					ST_Completing	:= FALSE;
					ST_Aborting		:= TRUE;
				ELSIF Stop THEN
					ePMLState 		:= E_PMLState.STOPPING;
					ST_Completing	:= FALSE;
					ST_Stopping		:= TRUE;
				ELSIF StateComplete AND NOT StateCompletePrev THEN
					ePMLState 		:= E_PMLState.COMPLETE;
					StateCompletePrev := StateComplete;
					ST_Completing	:= FALSE;
					ST_Complete		:= TRUE;
				END_IF


	E_PMLState.COMPLETE:
				(* final state *)
		
				IF bStateChange THEN
					(* transient state *)
					ST_Starting		:= FALSE;
					ST_Completing	:= FALSE;
					ST_Resetting	:= FALSE;
					ST_Holding		:= FALSE;
					ST_UnHolding	:= FALSE;
					ST_Suspending	:= FALSE;
					ST_UnSuspending	:= FALSE;
					ST_Clearing		:= FALSE;
					ST_Stopping		:= FALSE;
					ST_Aborting		:= FALSE;
		
					(* final state *)
					ST_Execute		:= FALSE;
					ST_Complete		:= TRUE;
					ST_Idle			:= FALSE;
					ST_Held			:= FALSE;
					ST_Suspended	:= FALSE;
					ST_Stopped		:= FALSE;
					ST_Aborted		:= FALSE;
				END_IF
		
				IF Abort THEN
					ePMLState 		:= E_PMLState.ABORTING;
					ST_Complete		:= FALSE;
					ST_Aborting		:= TRUE;
				ELSIF Stop THEN
					ePMLState 		:= E_PMLState.STOPPING;
					ST_Complete		:= FALSE;
					ST_Stopping		:= TRUE;
				ELSIF Reset THEN
					ePMLState 		:= E_PMLState.RESETTING;
					ST_Complete		:= FALSE;
					ST_Resetting	:= TRUE;
				END_IF


	E_PMLState.RESETTING:
				(* transient state *)
		
				IF bStateChange THEN
					(* transient state *)
					ST_Starting		:= FALSE;
					ST_Completing	:= FALSE;
					ST_Resetting	:= TRUE;
					ST_Holding		:= FALSE;
					ST_UnHolding	:= FALSE;
					ST_Suspending	:= FALSE;
					ST_UnSuspending	:= FALSE;
					ST_Clearing		:= FALSE;
					ST_Stopping		:= FALSE;
					ST_Aborting		:= FALSE;
		
					(* final state *)
					ST_Execute		:= FALSE;
					ST_Complete		:= FALSE;
					ST_Idle			:= FALSE;
					ST_Held			:= FALSE;
					ST_Suspended	:= FALSE;
					ST_Stopped		:= FALSE;
					ST_Aborted		:= FALSE;
				END_IF
		
				IF Abort THEN
					ePMLState 		:= E_PMLState.ABORTING;
					ST_Resetting	:= FALSE;
					ST_Aborting		:= TRUE;
				ELSIF Stop THEN
					ePMLState 		:= E_PMLState.STOPPING;
					ST_Resetting	:= FALSE;
					ST_Stopping		:= TRUE;
				ELSIF StateComplete THEN
					ePMLState 		:= E_PMLState.IDLE;
					StateCompletePrev := StateComplete;
					ST_Resetting	:= FALSE;
					ST_Idle			:= TRUE;
				END_IF


	E_PMLState.HOLDING:
				(* transient state *)
		
				IF bStateChange THEN
					(* transient state *)
					ST_Starting		:= FALSE;
					ST_Completing	:= FALSE;
					ST_Resetting	:= FALSE;
					ST_Holding		:= TRUE;
					ST_UnHolding	:= FALSE;
					ST_Suspending	:= FALSE;
					ST_UnSuspending	:= FALSE;
					ST_Clearing		:= FALSE;
					ST_Stopping		:= FALSE;
					ST_Aborting		:= FALSE;
		
					(* final state *)
					ST_Execute		:= FALSE;
					ST_Complete		:= FALSE;
					ST_Idle			:= FALSE;
					ST_Held			:= FALSE;
					ST_Suspended	:= FALSE;
					ST_Stopped		:= FALSE;
					ST_Aborted		:= FALSE;
				END_IF
		
				IF Abort THEN
					ePMLState 		:= E_PMLState.ABORTING;
					ST_Holding		:= FALSE;
					ST_Aborting		:= TRUE;
				ELSIF Stop THEN
					ePMLState 		:= E_PMLState.STOPPING;
					ST_Holding		:= FALSE;
					ST_Stopping		:= TRUE;
				ELSIF StateComplete AND NOT StateCompletePrev THEN
					ePMLState 		:= E_PMLState.HELD;
					StateCompletePrev := StateComplete;
					ST_Holding		:= FALSE;
					ST_Held			:= TRUE;
				END_IF


	E_PMLState.HELD:
				(* final state *)

				IF bStateChange THEN
					(* transient state *)
					ST_Starting		:= FALSE;
					ST_Completing	:= FALSE;
					ST_Resetting	:= FALSE;
					ST_Holding		:= FALSE;
					ST_UnHolding	:= FALSE;
					ST_Suspending	:= FALSE;
					ST_UnSuspending	:= FALSE;
					ST_Clearing		:= FALSE;
					ST_Stopping		:= FALSE;
					ST_Aborting		:= FALSE;
		
					(* final state *)
					ST_Execute		:= FALSE;
					ST_Complete		:= FALSE;
					ST_Idle			:= FALSE;
					ST_Held			:= TRUE;
					ST_Suspended	:= FALSE;
					ST_Stopped		:= FALSE;
					ST_Aborted		:= FALSE;
				END_IF
		
				IF Abort THEN
					ePMLState 		:= E_PMLState.ABORTING;
					ST_Held			:= FALSE;
					ST_Aborting		:= TRUE;
				ELSIF Stop THEN
					ePMLState 		:= E_PMLState.STOPPING;
					ST_Held			:= FALSE;
					ST_Stopping		:= TRUE;
				ELSIF UnHold THEN
					ePMLState 		:= E_PMLState.UNHOLDING;
					ST_Held			:= FALSE;
					ST_UnHolding	:= TRUE;
				END_IF


	E_PMLState.UNHOLDING:
				(* transient state *)
		
				IF bStateChange THEN
					(* transient state *)
					ST_Starting		:= FALSE;
					ST_Completing	:= FALSE;
					ST_Resetting	:= FALSE;
					ST_Holding		:= FALSE;
					ST_UnHolding	:= TRUE;
					ST_Suspending	:= FALSE;
					ST_UnSuspending	:= FALSE;
					ST_Clearing		:= FALSE;
					ST_Stopping		:= FALSE;
					ST_Aborting		:= FALSE;
		
					(* final state *)
					ST_Execute		:= FALSE;
					ST_Complete		:= FALSE;
					ST_Idle			:= FALSE;
					ST_Held			:= FALSE;
					ST_Suspended	:= FALSE;
					ST_Stopped		:= FALSE;
					ST_Aborted		:= FALSE;
				END_IF
		
				IF Abort THEN
					ePMLState 		:= E_PMLState.ABORTING;
					ST_UnHolding	:= FALSE;
					ST_Aborting		:= TRUE;
				ELSIF Stop THEN
					ePMLState 		:= E_PMLState.STOPPING;
					ST_UnHolding	:= FALSE;
					ST_Stopping		:= TRUE;
				ELSIF StateComplete AND NOT StateCompletePrev THEN
					ePMLState 		:= E_PMLState.EXECUTE;
					StateCompletePrev := StateComplete;
					ST_UnHolding	:= FALSE;
					ST_Execute		:= TRUE;
				END_IF


	E_PMLState.SUSPENDING:
				(* transient state *)
		
				IF bStateChange THEN
					(* transient state *)
					ST_Starting		:= FALSE;
					ST_Completing	:= FALSE;
					ST_Resetting	:= FALSE;
					ST_Holding		:= FALSE;
					ST_UnHolding	:= FALSE;
					ST_Suspending	:= TRUE;
					ST_UnSuspending	:= FALSE;
					ST_Clearing		:= FALSE;
					ST_Stopping		:= FALSE;
					ST_Aborting		:= FALSE;
		
					(* final state *)
					ST_Execute		:= FALSE;
					ST_Complete		:= FALSE;
					ST_Idle			:= FALSE;
					ST_Held			:= FALSE;
					ST_Suspended	:= FALSE;
					ST_Stopped		:= FALSE;
					ST_Aborted		:= FALSE;
				END_IF
		
				IF Abort THEN
					ePMLState 		:= E_PMLState.ABORTING;
					ST_Suspending	:= FALSE;
					ST_Aborting		:= TRUE;
				ELSIF Stop THEN
					ePMLState 		:= E_PMLState.STOPPING;
					ST_Suspending	:= FALSE;
					ST_Stopping		:= TRUE;
				ELSIF StateComplete AND NOT StateCompletePrev THEN
					ePMLState 		:= E_PMLState.SUSPENDED;
					StateCompletePrev := StateComplete;
					ST_Suspending	:= FALSE;
					ST_Suspended	:= TRUE;
				END_IF


	E_PMLState.SUSPENDED:
				(* final state *)
		
				IF bStateChange THEN
					(* transient state *)
					ST_Starting		:= FALSE;
					ST_Completing	:= FALSE;
					ST_Resetting	:= FALSE;
					ST_Holding		:= FALSE;
					ST_UnHolding	:= FALSE;
					ST_Suspending	:= FALSE;
					ST_UnSuspending	:= FALSE;
					ST_Clearing		:= FALSE;
					ST_Stopping		:= FALSE;
					ST_Aborting		:= FALSE;
		
					(* final state *)
					ST_Execute		:= FALSE;
					ST_Complete		:= FALSE;
					ST_Idle			:= FALSE;
					ST_Held			:= FALSE;
					ST_Suspended	:= TRUE;
					ST_Stopped		:= FALSE;
					ST_Aborted		:= FALSE;
				END_IF
		
				IF Abort THEN
					ePMLState 		:= E_PMLState.ABORTING;
					ST_Suspended	:= FALSE;
					ST_Aborting		:= TRUE;
				ELSIF Stop THEN
					ePMLState 		:= E_PMLState.STOPPING;
					ST_Suspended	:= FALSE;
					ST_Stopping		:= TRUE;
				ELSIF UnSuspend THEN
					ePMLState 		:= E_PMLState.UNSUSPENDING;
					ST_Suspended	:= FALSE;
					ST_UnSuspending	:= TRUE;
				END_IF


	E_PMLState.UNSUSPENDING:
				(* transient state *)
		
				IF bStateChange THEN
					(* transient state *)
					ST_Starting		:= FALSE;
					ST_Completing	:= FALSE;
					ST_Resetting	:= FALSE;
					ST_Holding		:= FALSE;
					ST_UnHolding	:= FALSE;
					ST_Suspending	:= FALSE;
					ST_UnSuspending	:= TRUE;
					ST_Clearing		:= FALSE;
					ST_Stopping		:= FALSE;
					ST_Aborting		:= FALSE;
		
					(* final state *)
					ST_Execute		:= FALSE;
					ST_Complete		:= FALSE;
					ST_Idle			:= FALSE;
					ST_Held			:= FALSE;
					ST_Suspended	:= FALSE;
					ST_Stopped		:= FALSE;
					ST_Aborted		:= FALSE;
				END_IF
		
				IF Abort THEN
					ePMLState 		:= E_PMLState.ABORTING;
					ST_UnSuspending	:= FALSE;
					ST_Aborting		:= TRUE;
				ELSIF Stop THEN
					ePMLState 		:= E_PMLState.STOPPING;
					ST_UnSuspending	:= FALSE;
					ST_Stopping		:= TRUE;
				ELSIF StateComplete AND NOT StateCompletePrev THEN
					ePMLState 		:= E_PMLState.EXECUTE;
					StateCompletePrev := StateComplete;
					ST_UnSuspending	:= FALSE;
					ST_Execute		:= TRUE;
				END_IF


	E_PMLState.STOPPING:
				(* transient state *)
		
				IF bStateChange THEN
					(* transient state *)
					ST_Starting		:= FALSE;
					ST_Completing	:= FALSE;
					ST_Resetting	:= FALSE;
					ST_Holding		:= FALSE;
					ST_UnHolding	:= FALSE;
					ST_Suspending	:= FALSE;
					ST_UnSuspending	:= FALSE;
					ST_Clearing		:= FALSE;
					ST_Stopping		:= TRUE;
					ST_Aborting		:= FALSE;
		
					(* final state *)
					ST_Execute		:= FALSE;
					ST_Complete		:= FALSE;
					ST_Idle			:= FALSE;
					ST_Held			:= FALSE;
					ST_Suspended	:= FALSE;
					ST_Stopped		:= FALSE;
					ST_Aborted		:= FALSE;
				END_IF
		
				IF Abort THEN
					ePMLState 		:= E_PMLState.ABORTING;
					ST_Stopping		:= FALSE;
					ST_Aborting		:= TRUE;
				ELSIF StateComplete AND NOT StateCompletePrev THEN
					ePMLState 		:= E_PMLState.STOPPED;
					StateCompletePrev := StateComplete;
					ST_Stopping		:= FALSE;
					ST_Stopped		:= TRUE;
				END_IF
				

	E_PMLState.STOPPED:
				(* final state *)
		
				IF bStateChange THEN
					(* transient state *)
					ST_Starting		:= FALSE;
					ST_Completing	:= FALSE;
					ST_Resetting	:= FALSE;
					ST_Holding		:= FALSE;
					ST_UnHolding	:= FALSE;
					ST_Suspending	:= FALSE;
					ST_UnSuspending	:= FALSE;
					ST_Clearing		:= FALSE;
					ST_Stopping		:= FALSE;
					ST_Aborting		:= FALSE;
		
					(* final state *)
					ST_Execute		:= FALSE;
					ST_Complete		:= FALSE;
					ST_Idle			:= FALSE;
					ST_Held			:= FALSE;
					ST_Suspended	:= FALSE;
					ST_Stopped		:= TRUE;
					ST_Aborted		:= FALSE;
				END_IF
		
				IF Abort THEN
					ePMLState 		:= E_PMLState.ABORTING;
					ST_Stopped		:= FALSE;
					ST_Aborting		:= TRUE;
				ELSIF Reset THEN
					ePMLState 		:= E_PMLState.RESETTING;
					ST_Stopped		:= FALSE;
					ST_Resetting	:= TRUE;
				END_IF


	E_PMLState.ABORTING:
				(* transient state *)
		
				IF bStateChange THEN
					(* transient state *)
					ST_Starting		:= FALSE;
					ST_Completing	:= FALSE;
					ST_Resetting	:= FALSE;
					ST_Holding		:= FALSE;
					ST_UnHolding	:= FALSE;
					ST_Suspending	:= FALSE;
					ST_UnSuspending	:= FALSE;
					ST_Clearing		:= FALSE;
					ST_Stopping		:= FALSE;
					ST_Aborting		:= TRUE;
		
					(* final state *)
					ST_Execute		:= FALSE;
					ST_Complete		:= FALSE;
					ST_Idle			:= FALSE;
					ST_Held			:= FALSE;
					ST_Suspended	:= FALSE;
					ST_Stopped		:= FALSE;
					ST_Aborted		:= FALSE;
				END_IF
		
				IF StateComplete AND NOT StateCompletePrev THEN
					ePMLState 		:= E_PMLState.ABORTED;
					StateCompletePrev := StateComplete;
					ST_Aborting		:= FALSE;
					ST_Aborted		:= TRUE;
				END_IF


	E_PMLState.ABORTED:
				(* final state *)
		
				IF bStateChange THEN
					(* transient state *)
					ST_Starting		:= FALSE;
					ST_Completing	:= FALSE;
					ST_Resetting	:= FALSE;
					ST_Holding		:= FALSE;
					ST_UnHolding	:= FALSE;
					ST_Suspending	:= FALSE;
					ST_UnSuspending	:= FALSE;
					ST_Clearing		:= FALSE;
					ST_Stopping		:= FALSE;
					ST_Aborting		:= FALSE;
		
					(* final state *)
					ST_Execute		:= FALSE;
					ST_Complete		:= FALSE;
					ST_Idle			:= FALSE;
					ST_Held			:= FALSE;
					ST_Suspended	:= FALSE;
					ST_Stopped		:= FALSE;
					ST_Aborted		:= TRUE;
				END_IF
		
				IF Clear THEN
					ePMLState 		:= E_PMLState.CLEARING;
					ST_Aborted		:= FALSE;
					ST_Clearing		:= TRUE;
				END_IF


	E_PMLState.CLEARING:
				(* transient state *)
		
				IF bStateChange THEN
					(* transient state *)
					ST_Starting		:= FALSE;
					ST_Completing	:= FALSE;
					ST_Resetting	:= FALSE;
					ST_Holding		:= FALSE;
					ST_UnHolding	:= FALSE;
					ST_Suspending	:= FALSE;
					ST_UnSuspending	:= FALSE;
					ST_Clearing		:= TRUE;
					ST_Stopping		:= FALSE;
					ST_Aborting		:= FALSE;
		
					(* final state *)
					ST_Execute		:= FALSE;
					ST_Complete		:= FALSE;
					ST_Idle			:= FALSE;
					ST_Held			:= FALSE;
					ST_Suspended	:= FALSE;
					ST_Stopped		:= FALSE;
					ST_Aborted		:= FALSE;
				END_IF
		
				IF Abort THEN
					ePMLState 		:= E_PMLState.ABORTING;
					ST_Stopped		:= FALSE;
					ST_Aborting		:= TRUE;
				ELSIF StateComplete AND NOT StateCompletePrev THEN
					ePMLState 		:= E_PMLState.STOPPED;
					StateCompletePrev := StateComplete;
					ST_Clearing		:= FALSE;
					ST_Stopped		:= TRUE;
				END_IF

END_CASE

(* auto clear with StateComplete = FALSE *)
StateCompletePrev := StateCompletePrev AND StateComplete;

END_FUNCTION_BLOCK

// ---- 00_Internal PackAL/POUs/PS_PackML_StateMachine_Maintenance.TcPOU
FUNCTION_BLOCK PS_PackML_StateMachine_Maintenance
VAR_INPUT
	Start				: BOOL;
	Hold				: BOOL;
	UnHold				: BOOL;
	Suspend				: BOOL;
	UnSuspend			: BOOL;
	Abort				: BOOL;
	Stop				: BOOL;
	Complete			: BOOL;
	Clear				: BOOL;
	Reset				: BOOL;
	StateComplete		: BOOL;
END_VAR
VAR_OUTPUT
	Status				: WORD;

	ST_Starting			: BOOL;
	ST_Completing		: BOOL;
	ST_Resetting		: BOOL;
	ST_Holding			: BOOL;
	ST_UnHolding		: BOOL;
	ST_Suspending		: BOOL;
	ST_UnSuspending		: BOOL;
	ST_Clearing			: BOOL;
	ST_Stopping			: BOOL;
	ST_Aborting			: BOOL;

	(* State Complete*)
	ST_Execute			: BOOL;
	ST_Complete			: BOOL;
	ST_Idle				: BOOL;
	ST_Held				: BOOL;
	ST_Suspended		: BOOL;
	ST_Stopped			: BOOL;
	ST_Aborted			: BOOL;

	(* additional *)
	Error				: BOOL;
	ErrorID				: DWORD;
	ePMLState			: E_PMLState := E_PMLState.IDLE;
END_VAR
VAR
	ePMLStatePrev		: E_PMLState;
	bStateChange		: BOOL;
	StateCompletePrev	: BOOL;
END_VAR

(* check for state change *)
IF ePMLStatePrev <> ePMLState THEN
	ePMLStatePrev 	:= ePMLState;
	bStateChange	:= TRUE;
ELSE
	bStateChange	:= FALSE;
END_IF


(* change to new state if requested *)
CASE ePMLState OF
	E_PMLState.UNDEFINED:
				(* undefined state *)
				IF bStateChange THEN
					(* transient state *)
					ST_Starting		:= FALSE;
					ST_Completing	:= FALSE;
					ST_Resetting	:= FALSE;
					ST_Holding		:= FALSE;
					ST_UnHolding	:= FALSE;
					ST_Suspending	:= FALSE;
					ST_UnSuspending	:= FALSE;
					ST_Clearing		:= FALSE;
					ST_Stopping		:= FALSE;
					ST_Aborting		:= FALSE;
		
					(* final state *)
					ST_Execute		:= FALSE;
					ST_Complete		:= FALSE;
					ST_Idle			:= FALSE;
					ST_Held			:= FALSE;
					ST_Suspended	:= FALSE;
					ST_Stopped		:= FALSE;
					ST_Aborted		:= FALSE;
				END_IF
		
				IF Abort THEN
					ePMLState 		:= E_PMLState.ABORTING;
					ST_Aborting		:= TRUE;
				ELSIF Stop THEN
					ePMLState 		:= E_PMLState.STOPPING;
					ST_Stopping		:= TRUE;
				END_IF


	E_PMLState.IDLE:
				(* final state *)
		
				IF bStateChange THEN
					(* transient state *)
					ST_Starting		:= FALSE;
					ST_Completing	:= FALSE;
					ST_Resetting	:= FALSE;
					ST_Holding		:= FALSE;
					ST_UnHolding	:= FALSE;
					ST_Suspending	:= FALSE;
					ST_UnSuspending	:= FALSE;
					ST_Clearing		:= FALSE;
					ST_Stopping		:= FALSE;
					ST_Aborting		:= FALSE;
		
					(* final state *)
					ST_Execute		:= FALSE;
					ST_Complete		:= FALSE;
					ST_Idle			:= TRUE;
					ST_Held			:= FALSE;
					ST_Suspended	:= FALSE;
					ST_Stopped		:= FALSE;
					ST_Aborted		:= FALSE;
				END_IF
		
				IF Abort THEN
					ePMLState 		:= E_PMLState.ABORTING;
					ST_Idle			:= FALSE;
					ST_Aborting		:= TRUE;
				ELSIF Stop THEN
					ePMLState 		:= E_PMLState.STOPPING;
					ST_Idle			:= FALSE;
					ST_Stopping		:= TRUE;
				ELSIF Start THEN
					ePMLState 		:= E_PMLState.STARTING;
					ST_Idle			:= FALSE;
					ST_Starting		:= TRUE;
				END_IF


	E_PMLState.STARTING:
				(* transient state *)
		
				IF bStateChange THEN
					(* transient state *)
					ST_Starting		:= TRUE;
					ST_Completing	:= FALSE;
					ST_Resetting	:= FALSE;
					ST_Holding		:= FALSE;
					ST_UnHolding	:= FALSE;
					ST_Suspending	:= FALSE;
					ST_UnSuspending	:= FALSE;
					ST_Clearing		:= FALSE;
					ST_Stopping		:= FALSE;
					ST_Aborting		:= FALSE;
		
					(* final state *)
					ST_Execute		:= FALSE;
					ST_Complete		:= FALSE;
					ST_Idle			:= FALSE;
					ST_Held			:= FALSE;
					ST_Suspended	:= FALSE;
					ST_Stopped		:= FALSE;
					ST_Aborted		:= FALSE;
				END_IF
		
				IF Abort THEN
					ePMLState 		:= E_PMLState.ABORTING;
					ST_Starting		:= FALSE;
					ST_Aborting		:= TRUE;
				ELSIF Stop THEN
					ePMLState 		:= E_PMLState.STOPPING;
					ST_Starting		:= FALSE;
					ST_Stopping		:= TRUE;
				ELSIF StateComplete AND NOT StateCompletePrev THEN
					ePMLState 		:= E_PMLState.EXECUTE;
					StateCompletePrev := StateComplete;
					ST_Starting		:= FALSE;
					ST_Execute		:= TRUE;
				END_IF


	E_PMLState.EXECUTE:
				(* final state *)
		
				IF bStateChange THEN
					(* transient state *)
					ST_Starting		:= FALSE;
					ST_Completing	:= FALSE;
					ST_Resetting	:= FALSE;
					ST_Holding		:= FALSE;
					ST_UnHolding	:= FALSE;
					ST_Suspending	:= FALSE;
					ST_UnSuspending	:= FALSE;
					ST_Clearing		:= FALSE;
					ST_Stopping		:= FALSE;
					ST_Aborting		:= FALSE;
		
					(* final state *)
					ST_Execute		:= TRUE;
					ST_Complete		:= FALSE;
					ST_Idle			:= FALSE;
					ST_Held			:= FALSE;
					ST_Suspended	:= FALSE;
					ST_Stopped		:= FALSE;
					ST_Aborted		:= FALSE;
				END_IF
		
				IF Abort THEN
					ePMLState 		:= E_PMLState.ABORTING;
					ST_Execute		:= FALSE;
					ST_Aborting		:= TRUE;
				ELSIF Stop THEN
					ePMLState 		:= E_PMLState.STOPPING;
					ST_Execute		:= FALSE;
					ST_Stopping		:= TRUE;
				ELSIF Hold THEN
					ePMLState 		:= E_PMLState.HOLDING;
					ST_Execute		:= FALSE;
					ST_Holding		:= TRUE;
				END_IF


	E_PMLState.RESETTING:
				(* transient state *)
		
				IF bStateChange THEN
					(* transient state *)
					ST_Starting		:= FALSE;
					ST_Completing	:= FALSE;
					ST_Resetting	:= TRUE;
					ST_Holding		:= FALSE;
					ST_UnHolding	:= FALSE;
					ST_Suspending	:= FALSE;
					ST_UnSuspending	:= FALSE;
					ST_Clearing		:= FALSE;
					ST_Stopping		:= FALSE;
					ST_Aborting		:= FALSE;
		
					(* final state *)
					ST_Execute		:= FALSE;
					ST_Complete		:= FALSE;
					ST_Idle			:= FALSE;
					ST_Held			:= FALSE;
					ST_Suspended	:= FALSE;
					ST_Stopped		:= FALSE;
					ST_Aborted		:= FALSE;
				END_IF
		
				IF Abort THEN
					ePMLState 		:= E_PMLState.ABORTING;
					ST_Resetting	:= FALSE;
					ST_Aborting		:= TRUE;
				ELSIF Stop THEN
					ePMLState 		:= E_PMLState.STOPPING;
					ST_Resetting	:= FALSE;
					ST_Stopping		:= TRUE;
				ELSIF StateComplete AND NOT StateCompletePrev THEN
					ePMLState 		:= E_PMLState.IDLE;
					StateCompletePrev := StateComplete;
					ST_Resetting	:= FALSE;
					ST_Idle			:= TRUE;
				END_IF


	E_PMLState.HOLDING:
				(* transient state *)
		
				IF bStateChange THEN
					(* transient state *)
					ST_Starting		:= FALSE;
					ST_Completing	:= FALSE;
					ST_Resetting	:= FALSE;
					ST_Holding		:= TRUE;
					ST_UnHolding	:= FALSE;
					ST_Suspending	:= FALSE;
					ST_UnSuspending	:= FALSE;
					ST_Clearing		:= FALSE;
					ST_Stopping		:= FALSE;
					ST_Aborting		:= FALSE;
		
					(* final state *)
					ST_Execute		:= FALSE;
					ST_Complete		:= FALSE;
					ST_Idle			:= FALSE;
					ST_Held			:= FALSE;
					ST_Suspended	:= FALSE;
					ST_Stopped		:= FALSE;
					ST_Aborted		:= FALSE;
				END_IF
		
				IF Abort THEN
					ePMLState 		:= E_PMLState.ABORTING;
					ST_Holding		:= FALSE;
					ST_Aborting		:= TRUE;
				ELSIF Stop THEN
					ePMLState 		:= E_PMLState.STOPPING;
					ST_Holding		:= FALSE;
					ST_Stopping		:= TRUE;
				ELSIF StateComplete AND NOT StateCompletePrev THEN
					ePMLState 		:= E_PMLState.HELD;
					StateCompletePrev := StateComplete;
					ST_Holding		:= FALSE;
					ST_Held			:= TRUE;
				END_IF


	E_PMLState.HELD:
				(* final state *)
		
				IF bStateChange THEN
					(* transient state *)
					ST_Starting		:= FALSE;
					ST_Completing	:= FALSE;
					ST_Resetting	:= FALSE;
					ST_Holding		:= FALSE;
					ST_UnHolding	:= FALSE;
					ST_Suspending	:= FALSE;
					ST_UnSuspending	:= FALSE;
					ST_Clearing		:= FALSE;
					ST_Stopping		:= FALSE;
					ST_Aborting		:= FALSE;
		
					(* final state *)
					ST_Execute		:= FALSE;
					ST_Complete		:= FALSE;
					ST_Idle			:= FALSE;
					ST_Held			:= TRUE;
					ST_Suspended	:= FALSE;
					ST_Stopped		:= FALSE;
					ST_Aborted		:= FALSE;
				END_IF
		
				IF Abort THEN
					ePMLState 		:= E_PMLState.ABORTING;
					ST_Held			:= FALSE;
					ST_Aborting		:= TRUE;
				ELSIF Stop THEN
					ePMLState 		:= E_PMLState.STOPPING;
					ST_Held			:= FALSE;
					ST_Stopping		:= TRUE;
				ELSIF UnHold THEN
					ePMLState 		:= E_PMLState.UNHOLDING;
					ST_Held			:= FALSE;
					ST_UnHolding	:= TRUE;
				END_IF


	E_PMLState.UNHOLDING:
				(* transient state *)
		
				IF bStateChange THEN
					(* transient state *)
					ST_Starting		:= FALSE;
					ST_Completing	:= FALSE;
					ST_Resetting	:= FALSE;
					ST_Holding		:= FALSE;
					ST_UnHolding	:= TRUE;
					ST_Suspending	:= FALSE;
					ST_UnSuspending	:= FALSE;
					ST_Clearing		:= FALSE;
					ST_Stopping		:= FALSE;
					ST_Aborting		:= FALSE;
		
					(* final state *)
					ST_Execute		:= FALSE;
					ST_Complete		:= FALSE;
					ST_Idle			:= FALSE;
					ST_Held			:= FALSE;
					ST_Suspended	:= FALSE;
					ST_Stopped		:= FALSE;
					ST_Aborted		:= FALSE;
				END_IF
		
				IF Abort THEN
					ePMLState 		:= E_PMLState.ABORTING;
					ST_UnHolding	:= FALSE;
					ST_Aborting		:= TRUE;
				ELSIF Stop THEN
					ePMLState 		:= E_PMLState.STOPPING;
					ST_UnHolding	:= FALSE;
					ST_Stopping		:= TRUE;
				ELSIF StateComplete THEN
					ePMLState 		:= E_PMLState.EXECUTE;
					StateCompletePrev := StateComplete;
					ST_UnHolding	:= FALSE;
					ST_Execute		:= TRUE;
				END_IF


	E_PMLState.STOPPING:
				(* transient state *)
		
				IF bStateChange THEN
					(* transient state *)
					ST_Starting		:= FALSE;
					ST_Completing	:= FALSE;
					ST_Resetting	:= FALSE;
					ST_Holding		:= FALSE;
					ST_UnHolding	:= FALSE;
					ST_Suspending	:= FALSE;
					ST_UnSuspending	:= FALSE;
					ST_Clearing		:= FALSE;
					ST_Stopping		:= TRUE;
					ST_Aborting		:= FALSE;
		
					(* final state *)
					ST_Execute		:= FALSE;
					ST_Complete		:= FALSE;
					ST_Idle			:= FALSE;
					ST_Held			:= FALSE;
					ST_Suspended	:= FALSE;
					ST_Stopped		:= FALSE;
					ST_Aborted		:= FALSE;
				END_IF
		
				IF Abort THEN
					ePMLState 		:= E_PMLState.ABORTING;
					ST_Stopping		:= FALSE;
					ST_Aborting		:= TRUE;
				ELSIF StateComplete AND NOT StateCompletePrev THEN
					ePMLState 		:= E_PMLState.STOPPED;
					StateCompletePrev := StateComplete;
					ST_Stopping		:= FALSE;
					ST_Stopped		:= TRUE;
				END_IF


	E_PMLState.STOPPED:
				(* final state *)
		
				IF bStateChange THEN
					(* transient state *)
					ST_Starting		:= FALSE;
					ST_Completing	:= FALSE;
					ST_Resetting	:= FALSE;
					ST_Holding		:= FALSE;
					ST_UnHolding	:= FALSE;
					ST_Suspending	:= FALSE;
					ST_UnSuspending	:= FALSE;
					ST_Clearing		:= FALSE;
					ST_Stopping		:= FALSE;
					ST_Aborting		:= FALSE;
		
					(* final state *)
					ST_Execute		:= FALSE;
					ST_Complete		:= FALSE;
					ST_Idle			:= FALSE;
					ST_Held			:= FALSE;
					ST_Suspended	:= FALSE;
					ST_Stopped		:= TRUE;
					ST_Aborted		:= FALSE;
				END_IF
		
				IF Abort THEN
					ePMLState 		:= E_PMLState.ABORTING;
					ST_Stopped		:= FALSE;
					ST_Aborting		:= TRUE;
				ELSIF Reset THEN
					ePMLState 		:= E_PMLState.RESETTING;
					ST_Stopped		:= FALSE;
					ST_Resetting	:= TRUE;
				END_IF


E_PMLState.ABORTING:
				(* transient state *)
		
				IF bStateChange THEN
					(* transient state *)
					ST_Starting		:= FALSE;
					ST_Completing	:= FALSE;
					ST_Resetting	:= FALSE;
					ST_Holding		:= FALSE;
					ST_UnHolding	:= FALSE;
					ST_Suspending	:= FALSE;
					ST_UnSuspending	:= FALSE;
					ST_Clearing		:= FALSE;
					ST_Stopping		:= FALSE;
					ST_Aborting		:= TRUE;
		
					(* final state *)
					ST_Execute		:= FALSE;
					ST_Complete		:= FALSE;
					ST_Idle			:= FALSE;
					ST_Held			:= FALSE;
					ST_Suspended	:= FALSE;
					ST_Stopped		:= FALSE;
					ST_Aborted		:= FALSE;
				END_IF
		
				IF StateComplete AND NOT StateCompletePrev THEN
					ePMLState 		:= E_PMLState.ABORTED;
					StateCompletePrev := StateComplete;
					ST_Aborting		:= FALSE;
					ST_Aborted		:= TRUE;
				END_IF


	E_PMLState.ABORTED:
				(* final state *)
		
				IF bStateChange THEN
					(* transient state *)
					ST_Starting		:= FALSE;
					ST_Completing	:= FALSE;
					ST_Resetting	:= FALSE;
					ST_Holding		:= FALSE;
					ST_UnHolding	:= FALSE;
					ST_Suspending	:= FALSE;
					ST_UnSuspending	:= FALSE;
					ST_Clearing		:= FALSE;
					ST_Stopping		:= FALSE;
					ST_Aborting		:= FALSE;
		
					(* final state *)
					ST_Execute		:= FALSE;
					ST_Complete		:= FALSE;
					ST_Idle			:= FALSE;
					ST_Held			:= FALSE;
					ST_Suspended	:= FALSE;
					ST_Stopped		:= FALSE;
					ST_Aborted		:= TRUE;
				END_IF
		
				IF Clear THEN
					ePMLState 		:= E_PMLState.CLEARING;
					ST_Aborted		:= FALSE;
					ST_Clearing		:= TRUE;
				END_IF


	E_PMLState.CLEARING:
				(* transient state *)
		
				IF bStateChange THEN
					(* transient state *)
					ST_Starting		:= FALSE;
					ST_Completing	:= FALSE;
					ST_Resetting	:= FALSE;
					ST_Holding		:= FALSE;
					ST_UnHolding	:= FALSE;
					ST_Suspending	:= FALSE;
					ST_UnSuspending	:= FALSE;
					ST_Clearing		:= TRUE;
					ST_Stopping		:= FALSE;
					ST_Aborting		:= FALSE;
		
					(* final state *)
					ST_Execute		:= FALSE;
					ST_Complete		:= FALSE;
					ST_Idle			:= FALSE;
					ST_Held			:= FALSE;
					ST_Suspended	:= FALSE;
					ST_Stopped		:= FALSE;
					ST_Aborted		:= FALSE;
				END_IF
		
				IF Abort THEN
					ePMLState 		:= E_PMLState.ABORTING;
					ST_Stopped		:= FALSE;
					ST_Aborting		:= TRUE;
				ELSIF StateComplete AND NOT StateCompletePrev THEN
					ePMLState 		:= E_PMLState.STOPPED;
					ST_Clearing		:= FALSE;
					ST_Stopped		:= TRUE;
				END_IF

END_CASE

(* auto clear with StateComplete = FALSE *)
StateCompletePrev := StateCompletePrev AND StateComplete;

END_FUNCTION_BLOCK

// ---- 00_Internal PackAL/POUs/PS_PackML_StateMachine_Manual.TcPOU
FUNCTION_BLOCK PS_PackML_StateMachine_Manual
VAR_INPUT
	Start				: BOOL;
	Hold				: BOOL;
	UnHold				: BOOL;
	Suspend				: BOOL;
	UnSuspend			: BOOL;
	Abort				: BOOL;
	Stop				: BOOL;
	Complete			: BOOL;
	Clear				: BOOL;
	Reset				: BOOL;
	StateComplete		: BOOL;
END_VAR
VAR_OUTPUT
	Status				: WORD;

	ST_Starting			: BOOL;
	ST_Completing		: BOOL;
	ST_Resetting		: BOOL;
	ST_Holding			: BOOL;
	ST_UnHolding		: BOOL;
	ST_Suspending		: BOOL;
	ST_UnSuspending		: BOOL;
	ST_Clearing			: BOOL;
	ST_Stopping			: BOOL;
	ST_Aborting			: BOOL;

	(* State Complete*)
	ST_Execute			: BOOL;
	ST_Complete			: BOOL;
	ST_Idle				: BOOL;
	ST_Held				: BOOL;
	ST_Suspended		: BOOL;
	ST_Stopped			: BOOL;
	ST_Aborted			: BOOL;

	(* additional *)
	Error				: BOOL;
	ErrorID				: DWORD;
	ePMLState			: E_PMLState := E_PMLState.IDLE;
END_VAR
VAR
	ePMLStatePrev		: E_PMLState;
	bStateChange		: BOOL;
	StateCompletePrev	: BOOL;
END_VAR

(* check for state change *)
IF ePMLStatePrev <> ePMLState THEN
	ePMLStatePrev 	:= ePMLState;
	bStateChange		:= TRUE;
ELSE
	bStateChange		:= FALSE;
END_IF


(* change to new state if requested *)
CASE ePMLState OF
	E_PMLState.UNDEFINED:
				(* undefined state *)
				IF bStateChange THEN
					(* transient state *)
					ST_Starting		:= FALSE;
					ST_Completing	:= FALSE;
					ST_Resetting	:= FALSE;
					ST_Holding		:= FALSE;
					ST_UnHolding	:= FALSE;
					ST_Suspending	:= FALSE;
					ST_UnSuspending	:= FALSE;
					ST_Clearing		:= FALSE;
					ST_Stopping		:= FALSE;
					ST_Aborting		:= FALSE;
		
					(* final state *)
					ST_Execute		:= FALSE;
					ST_Complete		:= FALSE;
					ST_Idle			:= FALSE;
					ST_Held			:= FALSE;
					ST_Suspended	:= FALSE;
					ST_Stopped		:= FALSE;
					ST_Aborted		:= FALSE;
				END_IF
		
				IF Abort THEN
					ePMLState 		:= E_PMLState.ABORTING;
					ST_Aborting		:= TRUE;
				ELSIF Stop THEN
					ePMLState 		:= E_PMLState.STOPPING;
					ST_Stopping		:= TRUE;
				END_IF


	E_PMLState.IDLE:
				(* final state *)
		
				IF bStateChange THEN
					(* transient state *)
					ST_Starting		:= FALSE;
					ST_Completing	:= FALSE;
					ST_Resetting	:= FALSE;
					ST_Holding		:= FALSE;
					ST_UnHolding	:= FALSE;
					ST_Suspending	:= FALSE;
					ST_UnSuspending	:= FALSE;
					ST_Clearing		:= FALSE;
					ST_Stopping		:= FALSE;
					ST_Aborting		:= FALSE;
		
					(* final state *)
					ST_Execute		:= FALSE;
					ST_Complete		:= FALSE;
					ST_Idle			:= TRUE;
					ST_Held			:= FALSE;
					ST_Suspended	:= FALSE;
					ST_Stopped		:= FALSE;
					ST_Aborted		:= FALSE;
				END_IF
		
				IF Abort THEN
					ePMLState 		:= E_PMLState.ABORTING;
					ST_Idle			:= FALSE;
					ST_Aborting		:= TRUE;
				ELSIF Stop THEN
					ePMLState 		:= E_PMLState.STOPPING;
					ST_Idle			:= FALSE;
					ST_Stopping		:= TRUE;
				ELSIF Start THEN
					ePMLState 		:= E_PMLState.STARTING;
					ST_Idle			:= FALSE;
					ST_Starting		:= TRUE;
				END_IF


	E_PMLState.STARTING:
				(* transient state *)
		
				IF bStateChange THEN
					(* transient state *)
					ST_Starting		:= TRUE;
					ST_Completing	:= FALSE;
					ST_Resetting	:= FALSE;
					ST_Holding		:= FALSE;
					ST_UnHolding	:= FALSE;
					ST_Suspending	:= FALSE;
					ST_UnSuspending	:= FALSE;
					ST_Clearing		:= FALSE;
					ST_Stopping		:= FALSE;
					ST_Aborting		:= FALSE;
		
					(* final state *)
					ST_Execute		:= FALSE;
					ST_Complete		:= FALSE;
					ST_Idle			:= FALSE;
					ST_Held			:= FALSE;
					ST_Suspended	:= FALSE;
					ST_Stopped		:= FALSE;
					ST_Aborted		:= FALSE;
				END_IF
		
				IF Abort THEN
					ePMLState 		:= E_PMLState.ABORTING;
					ST_Starting		:= FALSE;
					ST_Aborting		:= TRUE;
				ELSIF Stop THEN
					ePMLState 		:= E_PMLState.STOPPING;
					ST_Starting		:= FALSE;
					ST_Stopping		:= TRUE;
				ELSIF StateComplete AND NOT StateCompletePrev THEN
					ePMLState 		:= E_PMLState.EXECUTE;
					StateCompletePrev := StateComplete;
					ST_Starting		:= FALSE;
					ST_Execute		:= TRUE;
				END_IF


	E_PMLState.EXECUTE:
				(* final state *)
		
				IF bStateChange THEN
					(* transient state *)
					ST_Starting		:= FALSE;
					ST_Completing	:= FALSE;
					ST_Resetting	:= FALSE;
					ST_Holding		:= FALSE;
					ST_UnHolding	:= FALSE;
					ST_Suspending	:= FALSE;
					ST_UnSuspending	:= FALSE;
					ST_Clearing		:= FALSE;
					ST_Stopping		:= FALSE;
					ST_Aborting		:= FALSE;
		
					(* final state *)
					ST_Execute		:= TRUE;
					ST_Complete		:= FALSE;
					ST_Idle			:= FALSE;
					ST_Held			:= FALSE;
					ST_Suspended	:= FALSE;
					ST_Stopped		:= FALSE;
					ST_Aborted		:= FALSE;
				END_IF
		
				IF Abort THEN
					ePMLState 	:= E_PMLState.ABORTING;
					ST_Execute		:= FALSE;
					ST_Aborting		:= TRUE;
				ELSIF Stop THEN
					ePMLState 	:= E_PMLState.STOPPING;
					ST_Execute		:= FALSE;
					ST_Stopping		:= TRUE;
				END_IF


	E_PMLState.RESETTING:
				(* transient state *)
		
				IF bStateChange THEN
					(* transient state *)
					ST_Starting		:= FALSE;
					ST_Completing	:= FALSE;
					ST_Resetting	:= TRUE;
					ST_Holding		:= FALSE;
					ST_UnHolding	:= FALSE;
					ST_Suspending	:= FALSE;
					ST_UnSuspending	:= FALSE;
					ST_Clearing		:= FALSE;
					ST_Stopping		:= FALSE;
					ST_Aborting		:= FALSE;
		
					(* final state *)
					ST_Execute		:= FALSE;
					ST_Complete		:= FALSE;
					ST_Idle			:= FALSE;
					ST_Held			:= FALSE;
					ST_Suspended	:= FALSE;
					ST_Stopped		:= FALSE;
					ST_Aborted		:= FALSE;
				END_IF
		
				IF Abort THEN
					ePMLState 		:= E_PMLState.ABORTING;
					ST_Resetting	:= FALSE;
					ST_Aborting		:= TRUE;
				ELSIF Stop THEN
					ePMLState 		:= E_PMLState.STOPPING;
					ST_Resetting	:= FALSE;
					ST_Stopping		:= TRUE;
				ELSIF StateComplete AND NOT StateCompletePrev THEN
					ePMLState 		:= E_PMLState.IDLE;
					StateCompletePrev := StateComplete;
					ST_Resetting	:= FALSE;
					ST_Idle			:= TRUE;
				END_IF


	E_PMLState.STOPPING:
				(* transient state *)
		
				IF bStateChange THEN
					(* transient state *)
					ST_Starting		:= FALSE;
					ST_Completing	:= FALSE;
					ST_Resetting	:= FALSE;
					ST_Holding		:= FALSE;
					ST_UnHolding	:= FALSE;
					ST_Suspending	:= FALSE;
					ST_UnSuspending	:= FALSE;
					ST_Clearing		:= FALSE;
					ST_Stopping		:= TRUE;
					ST_Aborting		:= FALSE;
		
					(* final state *)
					ST_Execute		:= FALSE;
					ST_Complete		:= FALSE;
					ST_Idle			:= FALSE;
					ST_Held			:= FALSE;
					ST_Suspended	:= FALSE;
					ST_Stopped		:= FALSE;
					ST_Aborted		:= FALSE;
				END_IF
		
				IF Abort THEN
					ePMLState 		:= E_PMLState.ABORTING;
					ST_Stopping		:= FALSE;
					ST_Aborting		:= TRUE;
				ELSIF StateComplete AND NOT StateCompletePrev THEN
					ePMLState 		:= E_PMLState.STOPPED;
					StateCompletePrev := StateComplete;
					ST_Stopping		:= FALSE;
					ST_Stopped		:= TRUE;
				END_IF


	E_PMLState.STOPPED:
				(* final state *)
		
				IF bStateChange THEN
					(* transient state *)
					ST_Starting		:= FALSE;
					ST_Completing	:= FALSE;
					ST_Resetting	:= FALSE;
					ST_Holding		:= FALSE;
					ST_UnHolding	:= FALSE;
					ST_Suspending	:= FALSE;
					ST_UnSuspending	:= FALSE;
					ST_Clearing		:= FALSE;
					ST_Stopping		:= FALSE;
					ST_Aborting		:= FALSE;
		
					(* final state *)
					ST_Execute		:= FALSE;
					ST_Complete		:= FALSE;
					ST_Idle			:= FALSE;
					ST_Held			:= FALSE;
					ST_Suspended	:= FALSE;
					ST_Stopped		:= TRUE;
					ST_Aborted		:= FALSE;
				END_IF
		
				IF Abort THEN
					ePMLState 		:= E_PMLState.ABORTING;
					ST_Stopped		:= FALSE;
					ST_Aborting		:= TRUE;
				ELSIF Reset THEN
					ePMLState 		:= E_PMLState.RESETTING;
					ST_Stopped		:= FALSE;
					ST_Resetting	:= TRUE;
				END_IF


E_PMLState.ABORTING:
				(* transient state *)
		
				IF bStateChange THEN
					(* transient state *)
					ST_Starting		:= FALSE;
					ST_Completing	:= FALSE;
					ST_Resetting	:= FALSE;
					ST_Holding		:= FALSE;
					ST_UnHolding	:= FALSE;
					ST_Suspending	:= FALSE;
					ST_UnSuspending	:= FALSE;
					ST_Clearing		:= FALSE;
					ST_Stopping		:= FALSE;
					ST_Aborting		:= TRUE;
		
					(* final state *)
					ST_Execute		:= FALSE;
					ST_Complete		:= FALSE;
					ST_Idle			:= FALSE;
					ST_Held			:= FALSE;
					ST_Suspended	:= FALSE;
					ST_Stopped		:= FALSE;
					ST_Aborted		:= FALSE;
				END_IF
		
				IF StateComplete AND NOT StateCompletePrev THEN
					ePMLState 		:= E_PMLState.ABORTED;
					StateCompletePrev := StateComplete;
					ST_Aborting		:= FALSE;
					ST_Aborted		:= TRUE;
				END_IF


	E_PMLState.ABORTED:
				(* final state *)
		
				IF bStateChange THEN
					(* transient state *)
					ST_Starting		:= FALSE;
					ST_Completing	:= FALSE;
					ST_Resetting	:= FALSE;
					ST_Holding		:= FALSE;
					ST_UnHolding	:= FALSE;
					ST_Suspending	:= FALSE;
					ST_UnSuspending	:= FALSE;
					ST_Clearing		:= FALSE;
					ST_Stopping		:= FALSE;
					ST_Aborting		:= FALSE;
		
					(* final state *)
					ST_Execute		:= FALSE;
					ST_Complete		:= FALSE;
					ST_Idle			:= FALSE;
					ST_Held			:= FALSE;
					ST_Suspended	:= FALSE;
					ST_Stopped		:= FALSE;
					ST_Aborted		:= TRUE;
				END_IF
		
				IF Clear THEN
					ePMLState 	:= E_PMLState.CLEARING;
					ST_Aborted		:= FALSE;
					ST_Clearing		:= TRUE;
				END_IF


	E_PMLState.CLEARING:
				(* transient state *)
		
				IF bStateChange THEN
					(* transient state *)
					ST_Starting		:= FALSE;
					ST_Completing	:= FALSE;
					ST_Resetting	:= FALSE;
					ST_Holding		:= FALSE;
					ST_UnHolding	:= FALSE;
					ST_Suspending	:= FALSE;
					ST_UnSuspending	:= FALSE;
					ST_Clearing		:= TRUE;
					ST_Stopping		:= FALSE;
					ST_Aborting		:= FALSE;
		
					(* final state *)
					ST_Execute		:= FALSE;
					ST_Complete		:= FALSE;
					ST_Idle			:= FALSE;
					ST_Held			:= FALSE;
					ST_Suspended	:= FALSE;
					ST_Stopped		:= FALSE;
					ST_Aborted		:= FALSE;
				END_IF
		
				IF Abort THEN
					ePMLState 		:= E_PMLState.ABORTING;
					ST_Stopped		:= FALSE;
					ST_Aborting		:= TRUE;
				ELSIF StateComplete AND NOT StateCompletePrev THEN
					ePMLState 		:= E_PMLState.STOPPED;
					ST_Clearing		:= FALSE;
					ST_Stopped		:= TRUE;
				END_IF

END_CASE

(* auto clear with StateComplete = FALSE *)
StateCompletePrev := StateCompletePrev AND StateComplete;

END_FUNCTION_BLOCK

// ---- 00_Internal PackAL/POUs/PS_PackML_StateMachine_SemiAuto.TcPOU
FUNCTION_BLOCK PS_PackML_StateMachine_SemiAuto
VAR_INPUT
	Start				: BOOL;
	Hold				: BOOL;
	UnHold				: BOOL;
	Suspend				: BOOL;
	UnSuspend			: BOOL;
	Abort				: BOOL;
	Stop				: BOOL;
	Complete			: BOOL;
	Clear				: BOOL;
	Reset				: BOOL;
	StateComplete		: BOOL;
END_VAR
VAR_OUTPUT
	Status				: WORD;

	ST_Starting			: BOOL;
	ST_Completing		: BOOL;
	ST_Resetting		: BOOL;
	ST_Holding			: BOOL;
	ST_UnHolding		: BOOL;
	ST_Suspending		: BOOL;
	ST_UnSuspending		: BOOL;
	ST_Clearing			: BOOL;
	ST_Stopping			: BOOL;
	ST_Aborting			: BOOL;

	(* State Complete*)
	ST_Execute			: BOOL;
	ST_Complete			: BOOL;
	ST_Idle				: BOOL;
	ST_Held				: BOOL;
	ST_Suspended		: BOOL;
	ST_Stopped			: BOOL;
	ST_Aborted			: BOOL;

	(* additional *)
	Error				: BOOL;
	ErrorID				: DWORD;
	ePMLState			: E_PMLState := E_PMLState.IDLE;
END_VAR
VAR
	ePMLStatePrev		: E_PMLState;
	bStateChange		: BOOL;
	StateCompletePrev	: BOOL;
END_VAR

IF ePMLStatePrev <> ePMLState THEN
	ePMLStatePrev 	:= ePMLState;
	bStateChange	:= TRUE;
ELSE
	bStateChange	:= FALSE;
END_IF


(* change to new state if requested *)
CASE ePMLState OF
	E_PMLState.UNDEFINED:
				(* undefined state *)
				IF bStateChange THEN
					(* transient state *)
					ST_Starting		:= FALSE;
					ST_Completing	:= FALSE;
					ST_Resetting	:= FALSE;
					ST_Holding		:= FALSE;
					ST_UnHolding	:= FALSE;
					ST_Suspending	:= FALSE;
					ST_UnSuspending	:= FALSE;
					ST_Clearing		:= FALSE;
					ST_Stopping		:= FALSE;
					ST_Aborting		:= FALSE;
		
					(* final state *)
					ST_Execute		:= FALSE;
					ST_Complete		:= FALSE;
					ST_Idle			:= FALSE;
					ST_Held			:= FALSE;
					ST_Suspended	:= FALSE;
					ST_Stopped		:= FALSE;
					ST_Aborted		:= FALSE;
				END_IF
		
				IF Abort THEN
					ePMLState 		:= E_PMLState.ABORTING;
					ST_Aborting		:= TRUE;
				ELSIF Stop THEN
					ePMLState 		:= E_PMLState.STOPPING;
					ST_Stopping		:= TRUE;
				END_IF


	E_PMLState.IDLE:
				(* final state *)
		
				IF bStateChange THEN
					(* transient state *)
					ST_Starting		:= FALSE;
					ST_Completing	:= FALSE;
					ST_Resetting	:= FALSE;
					ST_Holding		:= FALSE;
					ST_UnHolding	:= FALSE;
					ST_Suspending	:= FALSE;
					ST_UnSuspending	:= FALSE;
					ST_Clearing		:= FALSE;
					ST_Stopping		:= FALSE;
					ST_Aborting		:= FALSE;
		
					(* final state *)
					ST_Execute		:= FALSE;
					ST_Complete		:= FALSE;
					ST_Idle			:= TRUE;
					ST_Held			:= FALSE;
					ST_Suspended	:= FALSE;
					ST_Stopped		:= FALSE;
					ST_Aborted		:= FALSE;
				END_IF
		
				IF Abort THEN
					ePMLState 	:= E_PMLState.ABORTING;
					ST_Idle			:= FALSE;
					ST_Aborting		:= TRUE;
				ELSIF Stop THEN
					ePMLState 	:= E_PMLState.STOPPING;
					ST_Idle			:= FALSE;
					ST_Stopping		:= TRUE;
				ELSIF Start THEN
					ePMLState 	:= E_PMLState.STARTING;
					ST_Idle			:= FALSE;
					ST_Starting		:= TRUE;
				END_IF


	E_PMLState.STARTING:
				(* transient state *)
		
				IF bStateChange THEN
					(* transient state *)
					ST_Starting		:= TRUE;
					ST_Completing	:= FALSE;
					ST_Resetting	:= FALSE;
					ST_Holding		:= FALSE;
					ST_UnHolding	:= FALSE;
					ST_Suspending	:= FALSE;
					ST_UnSuspending	:= FALSE;
					ST_Clearing		:= FALSE;
					ST_Stopping		:= FALSE;
					ST_Aborting		:= FALSE;
		
					(* final state *)
					ST_Execute		:= FALSE;
					ST_Complete		:= FALSE;
					ST_Idle			:= FALSE;
					ST_Held			:= FALSE;
					ST_Suspended	:= FALSE;
					ST_Stopped		:= FALSE;
					ST_Aborted		:= FALSE;
				END_IF
		
				IF Abort THEN
					ePMLState 		:= E_PMLState.ABORTING;
					ST_Starting		:= FALSE;
					ST_Aborting		:= TRUE;
				ELSIF Stop THEN
					ePMLState 		:= E_PMLState.STOPPING;
					ST_Starting		:= FALSE;
					ST_Stopping		:= TRUE;
				ELSIF StateComplete AND NOT StateCompletePrev THEN
					ePMLState 		:= E_PMLState.EXECUTE;
					StateCompletePrev := StateComplete;
					ST_Starting		:= FALSE;
					ST_Execute		:= TRUE;
				END_IF


	E_PMLState.EXECUTE:
				(* final state *)
		
				IF bStateChange THEN
					(* transient state *)
					ST_Starting		:= FALSE;
					ST_Completing	:= FALSE;
					ST_Resetting	:= FALSE;
					ST_Holding		:= FALSE;
					ST_UnHolding	:= FALSE;
					ST_Suspending	:= FALSE;
					ST_UnSuspending	:= FALSE;
					ST_Clearing		:= FALSE;
					ST_Stopping		:= FALSE;
					ST_Aborting		:= FALSE;
		
					(* final state *)
					ST_Execute		:= TRUE;
					ST_Complete		:= FALSE;
					ST_Idle			:= FALSE;
					ST_Held			:= FALSE;
					ST_Suspended	:= FALSE;
					ST_Stopped		:= FALSE;
					ST_Aborted		:= FALSE;
				END_IF
		
				IF Abort THEN
					ePMLState 		:= E_PMLState.ABORTING;
					ST_Execute		:= FALSE;
					ST_Aborting		:= TRUE;
				ELSIF Stop THEN
					ePMLState 		:= E_PMLState.STOPPING;
					ST_Execute		:= FALSE;
					ST_Stopping		:= TRUE;
				ELSIF Suspend THEN
					ePMLState 		:= E_PMLState.SUSPENDING;
					ST_Execute		:= FALSE;
					ST_Suspending	:= TRUE;
				ELSIF Hold THEN
					ePMLState 		:= E_PMLState.HOLDING;
					ST_Execute		:= FALSE;
					ST_Holding		:= TRUE;
				ELSIF Complete THEN
					ePMLState 		:= E_PMLState.COMPLETING;
					ST_Execute		:= FALSE;
					ST_Completing	:= TRUE;
				END_IF


	E_PMLState.COMPLETING:
				(* transient state *)
		
				IF bStateChange THEN
					(* transient state *)
					ST_Starting		:= FALSE;
					ST_Completing	:= TRUE;
					ST_Resetting	:= FALSE;
					ST_Holding		:= FALSE;
					ST_UnHolding	:= FALSE;
					ST_Suspending	:= FALSE;
					ST_UnSuspending	:= FALSE;
					ST_Clearing		:= FALSE;
					ST_Stopping		:= FALSE;
					ST_Aborting		:= FALSE;
		
					(* final state *)
					ST_Execute		:= FALSE;
					ST_Complete		:= FALSE;
					ST_Idle			:= FALSE;
					ST_Held			:= FALSE;
					ST_Suspended	:= FALSE;
					ST_Stopped		:= FALSE;
					ST_Aborted		:= FALSE;
				END_IF
		
				IF Abort THEN
					ePMLState 		:= E_PMLState.ABORTING;
					ST_Completing	:= FALSE;
					ST_Aborting		:= TRUE;
				ELSIF Stop THEN
					ePMLState 		:= E_PMLState.STOPPING;
					ST_Completing	:= FALSE;
					ST_Stopping		:= TRUE;
				ELSIF StateComplete AND NOT StateCompletePrev THEN
					ePMLState 		:= E_PMLState.COMPLETE;
					StateCompletePrev := StateComplete;
					ST_Completing	:= FALSE;
					ST_Complete		:= TRUE;
				END_IF


	E_PMLState.COMPLETE:
				(* final state *)
		
				IF bStateChange THEN
					(* transient state *)
					ST_Starting		:= FALSE;
					ST_Completing	:= FALSE;
					ST_Resetting	:= FALSE;
					ST_Holding		:= FALSE;
					ST_UnHolding	:= FALSE;
					ST_Suspending	:= FALSE;
					ST_UnSuspending	:= FALSE;
					ST_Clearing		:= FALSE;
					ST_Stopping		:= FALSE;
					ST_Aborting		:= FALSE;
		
					(* final state *)
					ST_Execute		:= FALSE;
					ST_Complete		:= TRUE;
					ST_Idle			:= FALSE;
					ST_Held			:= FALSE;
					ST_Suspended	:= FALSE;
					ST_Stopped		:= FALSE;
					ST_Aborted		:= FALSE;
				END_IF
		
				IF Abort THEN
					ePMLState 		:= E_PMLState.ABORTING;
					ST_Complete		:= FALSE;
					ST_Aborting		:= TRUE;
				ELSIF Stop THEN
					ePMLState 		:= E_PMLState.STOPPING;
					ST_Complete		:= FALSE;
					ST_Stopping		:= TRUE;
				ELSIF Reset THEN
					ePMLState 		:= E_PMLState.RESETTING;
					ST_Complete		:= FALSE;
					ST_Resetting	:= TRUE;
				END_IF


	E_PMLState.RESETTING:
				(* transient state *)
		
				IF bStateChange THEN
					(* transient state *)
					ST_Starting		:= FALSE;
					ST_Completing	:= FALSE;
					ST_Resetting	:= TRUE;
					ST_Holding		:= FALSE;
					ST_UnHolding	:= FALSE;
					ST_Suspending	:= FALSE;
					ST_UnSuspending	:= FALSE;
					ST_Clearing		:= FALSE;
					ST_Stopping		:= FALSE;
					ST_Aborting		:= FALSE;
		
					(* final state *)
					ST_Execute		:= FALSE;
					ST_Complete		:= FALSE;
					ST_Idle			:= FALSE;
					ST_Held			:= FALSE;
					ST_Suspended	:= FALSE;
					ST_Stopped		:= FALSE;
					ST_Aborted		:= FALSE;
				END_IF
		
				IF Abort THEN
					ePMLState 		:= E_PMLState.ABORTING;
					ST_Resetting	:= FALSE;
					ST_Aborting		:= TRUE;
				ELSIF Stop THEN
					ePMLState 		:= E_PMLState.STOPPING;
					ST_Resetting	:= FALSE;
					ST_Stopping		:= TRUE;
				ELSIF StateComplete AND NOT StateCompletePrev THEN
					ePMLState 		:= E_PMLState.IDLE;
					StateCompletePrev := StateComplete;
					ST_Resetting	:= FALSE;
					ST_Idle			:= TRUE;
				END_IF


	E_PMLState.HOLDING:
				(* transient state *)
		
				IF bStateChange THEN
					(* transient state *)
					ST_Starting		:= FALSE;
					ST_Completing	:= FALSE;
					ST_Resetting	:= FALSE;
					ST_Holding		:= TRUE;
					ST_UnHolding	:= FALSE;
					ST_Suspending	:= FALSE;
					ST_UnSuspending	:= FALSE;
					ST_Clearing		:= FALSE;
					ST_Stopping		:= FALSE;
					ST_Aborting		:= FALSE;
		
					(* final state *)
					ST_Execute		:= FALSE;
					ST_Complete		:= FALSE;
					ST_Idle			:= FALSE;
					ST_Held			:= FALSE;
					ST_Suspended	:= FALSE;
					ST_Stopped		:= FALSE;
					ST_Aborted		:= FALSE;
				END_IF
		
				IF Abort THEN
					ePMLState 		:= E_PMLState.ABORTING;
					ST_Holding		:= FALSE;
					ST_Aborting		:= TRUE;
				ELSIF Stop THEN
					ePMLState 		:= E_PMLState.STOPPING;
					ST_Holding		:= FALSE;
					ST_Stopping		:= TRUE;
				ELSIF StateComplete AND NOT StateCompletePrev THEN
					ePMLState 		:= E_PMLState.HELD;
					StateCompletePrev := StateComplete;
					ST_Holding		:= FALSE;
					ST_Held			:= TRUE;
				END_IF


	E_PMLState.HELD:
				(* final state *)
		
				IF bStateChange THEN
					(* transient state *)
					ST_Starting		:= FALSE;
					ST_Completing	:= FALSE;
					ST_Resetting	:= FALSE;
					ST_Holding		:= FALSE;
					ST_UnHolding	:= FALSE;
					ST_Suspending	:= FALSE;
					ST_UnSuspending	:= FALSE;
					ST_Clearing		:= FALSE;
					ST_Stopping		:= FALSE;
					ST_Aborting		:= FALSE;
		
					(* final state *)
					ST_Execute		:= FALSE;
					ST_Complete		:= FALSE;
					ST_Idle			:= FALSE;
					ST_Held			:= TRUE;
					ST_Suspended	:= FALSE;
					ST_Stopped		:= FALSE;
					ST_Aborted		:= FALSE;
				END_IF
		
				IF Abort THEN
					ePMLState 		:= E_PMLState.ABORTING;
					ST_Held			:= FALSE;
					ST_Aborting		:= TRUE;
				ELSIF Stop THEN
					ePMLState 		:= E_PMLState.STOPPING;
					ST_Held			:= FALSE;
					ST_Stopping		:= TRUE;
				ELSIF UnHold THEN
					ePMLState 		:= E_PMLState.UNHOLDING;
					ST_Held			:= FALSE;
					ST_UnHolding	:= TRUE;
				END_IF


	E_PMLState.UNHOLDING:
				(* transient state *)
		
				IF bStateChange THEN
					(* transient state *)
					ST_Starting		:= FALSE;
					ST_Completing	:= FALSE;
					ST_Resetting	:= FALSE;
					ST_Holding		:= FALSE;
					ST_UnHolding	:= TRUE;
					ST_Suspending	:= FALSE;
					ST_UnSuspending	:= FALSE;
					ST_Clearing		:= FALSE;
					ST_Stopping		:= FALSE;
					ST_Aborting		:= FALSE;
		
					(* final state *)
					ST_Execute		:= FALSE;
					ST_Complete		:= FALSE;
					ST_Idle			:= FALSE;
					ST_Held			:= FALSE;
					ST_Suspended	:= FALSE;
					ST_Stopped		:= FALSE;
					ST_Aborted		:= FALSE;
				END_IF
		
				IF Abort THEN
					ePMLState 		:= E_PMLState.ABORTING;
					ST_UnHolding	:= FALSE;
					ST_Aborting		:= TRUE;
				ELSIF Stop THEN
					ePMLState 		:= E_PMLState.STOPPING;
					ST_UnHolding	:= FALSE;
					ST_Stopping		:= TRUE;
				ELSIF StateComplete AND NOT StateCompletePrev THEN
					ePMLState 		:= E_PMLState.EXECUTE;
					StateCompletePrev := StateComplete;
					ST_UnHolding	:= FALSE;
					ST_Execute		:= TRUE;
				END_IF


	E_PMLState.SUSPENDING:
				(* transient state *)
		
				IF bStateChange THEN
					(* transient state *)
					ST_Starting		:= FALSE;
					ST_Completing	:= FALSE;
					ST_Resetting	:= FALSE;
					ST_Holding		:= FALSE;
					ST_UnHolding	:= FALSE;
					ST_Suspending	:= TRUE;
					ST_UnSuspending	:= FALSE;
					ST_Clearing		:= FALSE;
					ST_Stopping		:= FALSE;
					ST_Aborting		:= FALSE;
		
					(* final state *)
					ST_Execute		:= FALSE;
					ST_Complete		:= FALSE;
					ST_Idle			:= FALSE;
					ST_Held			:= FALSE;
					ST_Suspended	:= FALSE;
					ST_Stopped		:= FALSE;
					ST_Aborted		:= FALSE;
				END_IF
		
				IF Abort THEN
					ePMLState 		:= E_PMLState.ABORTING;
					ST_Suspending	:= FALSE;
					ST_Aborting		:= TRUE;
				ELSIF Stop THEN
					ePMLState 		:= E_PMLState.STOPPING;
					ST_Suspending	:= FALSE;
					ST_Stopping		:= TRUE;
				ELSIF StateComplete AND NOT StateCompletePrev THEN
					ePMLState 		:= E_PMLState.SUSPENDED;
					StateCompletePrev := StateComplete;
					ST_Suspending	:= FALSE;
					ST_Suspended	:= TRUE;
				END_IF


	E_PMLState.SUSPENDED:
				(* final state *)
		
				IF bStateChange THEN
					(* transient state *)
					ST_Starting		:= FALSE;
					ST_Completing	:= FALSE;
					ST_Resetting	:= FALSE;
					ST_Holding		:= FALSE;
					ST_UnHolding	:= FALSE;
					ST_Suspending	:= FALSE;
					ST_UnSuspending	:= FALSE;
					ST_Clearing		:= FALSE;
					ST_Stopping		:= FALSE;
					ST_Aborting		:= FALSE;
		
					(* final state *)
					ST_Execute		:= FALSE;
					ST_Complete		:= FALSE;
					ST_Idle			:= FALSE;
					ST_Held			:= FALSE;
					ST_Suspended	:= TRUE;
					ST_Stopped		:= FALSE;
					ST_Aborted		:= FALSE;
				END_IF
		
				IF Abort THEN
					ePMLState 		:= E_PMLState.ABORTING;
					ST_Suspended	:= FALSE;
					ST_Aborting		:= TRUE;
				ELSIF Stop THEN
					ePMLState 		:= E_PMLState.STOPPING;
					ST_Suspended	:= FALSE;
					ST_Stopping		:= TRUE;
				ELSIF UnSuspend THEN
					ePMLState 		:= E_PMLState.UNSUSPENDING;
					ST_Suspended	:= FALSE;
					ST_UnSuspending	:= TRUE;
				END_IF


	E_PMLState.UNSUSPENDING:
				(* transient state *)
		
				IF bStateChange THEN
					(* transient state *)
					ST_Starting		:= FALSE;
					ST_Completing	:= FALSE;
					ST_Resetting	:= FALSE;
					ST_Holding		:= FALSE;
					ST_UnHolding	:= FALSE;
					ST_Suspending	:= FALSE;
					ST_UnSuspending	:= TRUE;
					ST_Clearing		:= FALSE;
					ST_Stopping		:= FALSE;
					ST_Aborting		:= FALSE;
		
					(* final state *)
					ST_Execute		:= FALSE;
					ST_Complete		:= FALSE;
					ST_Idle			:= FALSE;
					ST_Held			:= FALSE;
					ST_Suspended	:= FALSE;
					ST_Stopped		:= FALSE;
					ST_Aborted		:= FALSE;
				END_IF
		
				IF Abort THEN
					ePMLState 		:= E_PMLState.ABORTING;
					ST_UnSuspending	:= FALSE;
					ST_Aborting		:= TRUE;
				ELSIF Stop THEN
					ePMLState 		:= E_PMLState.STOPPING;
					ST_UnSuspending	:= FALSE;
					ST_Stopping		:= TRUE;
				ELSIF StateComplete AND NOT StateCompletePrev THEN
					ePMLState 		:= E_PMLState.EXECUTE;
					StateCompletePrev := StateComplete;
					ST_UnSuspending	:= FALSE;
					ST_Execute		:= TRUE;
				END_IF


	E_PMLState.STOPPING:
				(* transient state *)
		
				IF bStateChange THEN
					(* transient state *)
					ST_Starting		:= FALSE;
					ST_Completing	:= FALSE;
					ST_Resetting	:= FALSE;
					ST_Holding		:= FALSE;
					ST_UnHolding	:= FALSE;
					ST_Suspending	:= FALSE;
					ST_UnSuspending	:= FALSE;
					ST_Clearing		:= FALSE;
					ST_Stopping		:= TRUE;
					ST_Aborting		:= FALSE;
		
					(* final state *)
					ST_Execute		:= FALSE;
					ST_Complete		:= FALSE;
					ST_Idle			:= FALSE;
					ST_Held			:= FALSE;
					ST_Suspended	:= FALSE;
					ST_Stopped		:= FALSE;
					ST_Aborted		:= FALSE;
				END_IF
		
				IF Abort THEN
					ePMLState 		:= E_PMLState.ABORTING;
					ST_Stopping		:= FALSE;
					ST_Aborting		:= TRUE;
				ELSIF StateComplete AND NOT StateCompletePrev THEN
					ePMLState 		:= E_PMLState.STOPPED;
					StateCompletePrev := StateComplete;
					ST_Stopping		:= FALSE;
					ST_Stopped		:= TRUE;
				END_IF


	E_PMLState.STOPPED:
				(* final state *)
		
				IF bStateChange THEN
					(* transient state *)
					ST_Starting		:= FALSE;
					ST_Completing	:= FALSE;
					ST_Resetting	:= FALSE;
					ST_Holding		:= FALSE;
					ST_UnHolding	:= FALSE;
					ST_Suspending	:= FALSE;
					ST_UnSuspending	:= FALSE;
					ST_Clearing		:= FALSE;
					ST_Stopping		:= FALSE;
					ST_Aborting		:= FALSE;
		
					(* final state *)
					ST_Execute		:= FALSE;
					ST_Complete		:= FALSE;
					ST_Idle			:= FALSE;
					ST_Held			:= FALSE;
					ST_Suspended	:= FALSE;
					ST_Stopped		:= TRUE;
					ST_Aborted		:= FALSE;
				END_IF
		
				IF Abort THEN
					ePMLState 		:= E_PMLState.ABORTING;
					ST_Stopped		:= FALSE;
					ST_Aborting		:= TRUE;
				ELSIF Reset THEN
					ePMLState 		:= E_PMLState.RESETTING;
					ST_Stopped		:= FALSE;
					ST_Resetting	:= TRUE;
				END_IF


E_PMLState.ABORTING:
				(* transient state *)
		
				IF bStateChange THEN
					(* transient state *)
					ST_Starting		:= FALSE;
					ST_Completing	:= FALSE;
					ST_Resetting	:= FALSE;
					ST_Holding		:= FALSE;
					ST_UnHolding	:= FALSE;
					ST_Suspending	:= FALSE;
					ST_UnSuspending	:= FALSE;
					ST_Clearing		:= FALSE;
					ST_Stopping		:= FALSE;
					ST_Aborting		:= TRUE;
		
					(* final state *)
					ST_Execute		:= FALSE;
					ST_Complete		:= FALSE;
					ST_Idle			:= FALSE;
					ST_Held			:= FALSE;
					ST_Suspended	:= FALSE;
					ST_Stopped		:= FALSE;
					ST_Aborted		:= FALSE;
				END_IF
		
				IF StateComplete AND NOT StateCompletePrev THEN
					ePMLState 		:= E_PMLState.ABORTED;
					StateCompletePrev := StateComplete;
					ST_Aborting		:= FALSE;
					ST_Aborted		:= TRUE;
				END_IF


	E_PMLState.ABORTED:
				(* final state *)
		
				IF bStateChange THEN
					(* transient state *)
					ST_Starting		:= FALSE;
					ST_Completing	:= FALSE;
					ST_Resetting	:= FALSE;
					ST_Holding		:= FALSE;
					ST_UnHolding	:= FALSE;
					ST_Suspending	:= FALSE;
					ST_UnSuspending	:= FALSE;
					ST_Clearing		:= FALSE;
					ST_Stopping		:= FALSE;
					ST_Aborting		:= FALSE;
		
					(* final state *)
					ST_Execute		:= FALSE;
					ST_Complete		:= FALSE;
					ST_Idle			:= FALSE;
					ST_Held			:= FALSE;
					ST_Suspended	:= FALSE;
					ST_Stopped		:= FALSE;
					ST_Aborted		:= TRUE;
				END_IF
		
				IF Clear THEN
					ePMLState 		:= E_PMLState.CLEARING;
					ST_Aborted		:= FALSE;
					ST_Clearing		:= TRUE;
				END_IF


	E_PMLState.CLEARING:
				(* transient state *)
		
				IF bStateChange THEN
					(* transient state *)
					ST_Starting		:= FALSE;
					ST_Completing	:= FALSE;
					ST_Resetting	:= FALSE;
					ST_Holding		:= FALSE;
					ST_UnHolding	:= FALSE;
					ST_Suspending	:= FALSE;
					ST_UnSuspending	:= FALSE;
					ST_Clearing		:= TRUE;
					ST_Stopping		:= FALSE;
					ST_Aborting		:= FALSE;
		
					(* final state *)
					ST_Execute		:= FALSE;
					ST_Complete		:= FALSE;
					ST_Idle			:= FALSE;
					ST_Held			:= FALSE;
					ST_Suspended	:= FALSE;
					ST_Stopped		:= FALSE;
					ST_Aborted		:= FALSE;
				END_IF
		
				IF Abort THEN
					ePMLState 		:= E_PMLState.ABORTING;
					ST_Stopped		:= FALSE;
					ST_Aborting		:= TRUE;
				ELSIF StateComplete AND NOT StateCompletePrev THEN
					ePMLState 		:= E_PMLState.STOPPED;
					StateCompletePrev := StateComplete;
					ST_Clearing		:= FALSE;
					ST_Stopped		:= TRUE;
				END_IF

END_CASE

(* auto clear with StateComplete = FALSE *)
StateCompletePrev := StateCompletePrev AND StateComplete;

END_FUNCTION_BLOCK

// ---- 00_Internal PackAL/POUs/PS_UnitModeManager.TcPOU
FUNCTION_BLOCK PS_UnitModeManager
VAR_INPUT
	Execute 		: BOOL;
	eModeCommand 	: E_PMLUnitMode;
	ePMLState		: E_PMLState;
END_VAR
VAR_OUTPUT
	eModeStatus 	: E_PMLUnitMode;
	Done 			: BOOL;
	Error 			: BOOL;
	ErrorID 		: UDINT;
END_VAR
VAR
	fbTrigger		: R_TRIG;
END_VAR

fbTrigger(CLK := Execute);

IF fbTrigger.Q THEN (* rising edge Execute *)
	Done 		:= FALSE;
	Error 		:= FALSE;
	ErrorID 	:= 0;

     CASE eModeStatus OF
		E_PMLUnitMode.UNDEFINED:
					eModeStatus := eModeCommand;
					Done := TRUE;

		E_PMLUnitMode.AUTOMATIC:
					IF (ePMLState = E_PMLState.STOPPED) OR (ePMLState = E_PMLState.ABORTED) OR (ePMLState = E_PMLState.IDLE) THEN
						eModeStatus := eModeCommand;
						Done := TRUE;
					ELSIF ((ePMLState = E_PMLState.SUSPENDED) OR (ePMLState = E_PMLState.HELD) OR (ePMLState = E_PMLState.COMPLETE))
						AND (eModeCommand = E_PMLUnitMode.SEMIAUTOMATIC) THEN
		
						eModeStatus := eModeCommand;
						Done := TRUE;
					ELSIF (ePMLState = E_PMLState.HELD) AND (eModeCommand = E_PMLUnitMode.MAINTENANCE) THEN
						eModeStatus := eModeCommand;
						Done := TRUE;
					ELSE
						Error := TRUE;
						ErrorID := 1;
					END_IF

		E_PMLUnitMode.MAINTENANCE:
					IF (ePMLState = E_PMLState.STOPPED) OR (ePMLState = E_PMLState.ABORTED) OR (ePMLState = E_PMLState.IDLE) THEN
						eModeStatus := eModeCommand;
						Done := TRUE;
					ELSIF (ePMLState = E_PMLState.HELD) AND ((eModeCommand = E_PMLUnitMode.AUTOMATIC) OR (eModeCommand = E_PMLUnitMode.SEMIAUTOMATIC)) THEN
						eModeStatus := eModeCommand;
						Done := TRUE;
					ELSE
						Error := TRUE;
						ErrorID := 1;
					END_IF

		E_PMLUnitMode.MANUAL:
					IF (ePMLState = E_PMLState.STOPPED) OR (ePMLState = E_PMLState.ABORTED) OR (ePMLState = E_PMLState.IDLE) THEN
						eModeStatus := eModeCommand;
						Done := TRUE;
					ELSE
						Error := TRUE;
						ErrorID := 1;
					END_IF

		E_PMLUnitMode.SEMIAUTOMATIC:
					IF (ePMLState = E_PMLState.STOPPED) OR (ePMLState = E_PMLState.ABORTED) OR (ePMLState = E_PMLState.IDLE) THEN
						eModeStatus := eModeCommand;
						Done := TRUE;
					ELSIF ((ePMLState = E_PMLState.SUSPENDED) OR (ePMLState = E_PMLState.HELD) OR (ePMLState = E_PMLState.COMPLETE))
						AND (eModeCommand = E_PMLUnitMode.AUTOMATIC) THEN
		
						eModeStatus := eModeCommand;
						Done := TRUE;
					ELSIF (ePMLState = E_PMLState.HELD) AND (eModeCommand = E_PMLUnitMode.MAINTENANCE) THEN
						eModeStatus := eModeCommand;
						Done := TRUE;
					ELSE
						Error := TRUE;
						ErrorID := 1;
					END_IF

		E_PMLUnitMode.DRYRUN:
					eModeStatus := eModeCommand;
					Done 		:= TRUE;

		E_PMLUnitMode.USERMODE1:
					eModeStatus := eModeCommand;
					Done 		:= TRUE;

		E_PMLUnitMode.USERMODE2:
					eModeStatus := eModeCommand;
					Done 		:= TRUE;

		E_PMLUnitMode.IDLE:
					IF (ePMLState = E_PMLState.STOPPED) OR (ePMLState = E_PMLState.ABORTED) OR (ePMLState = E_PMLState.IDLE) THEN
						eModeStatus := eModeCommand;
						Done 		:= TRUE;
					ELSE
						Error 	:= TRUE;
						ErrorID := 1;
					END_IF

		E_PMLUnitMode.ESTOP:
					IF (ePMLState = E_PMLState.STOPPED) OR (ePMLState = E_PMLState.ABORTED) OR (ePMLState = E_PMLState.IDLE) THEN
						 eModeStatus := eModeCommand;
						 Done 		:= TRUE;
					ELSE
						 Error 	:= TRUE;
						 ErrorID := 1;
					END_IF
     END_CASE
END_IF

 (* reset with bExecute = FALSE *)
 IF NOT Execute THEN
     Done 		:= FALSE;
     Error 		:= FALSE;
     ErrorID 	:= 0;
 END_IF

END_FUNCTION_BLOCK

// ---- 01_Submodules/FB_Axis.TcPOU
FUNCTION_BLOCK FB_Axis
VAR_OUTPUT
	// =============== State variables ========================
	bError			: BOOL;					// Error signal
	nErrorID		: UDINT;				// Error ID
	bMoves			: BOOL;					// Status of moving
END_VAR
VAR	
	// =============== Done signals of Halt and Reset =========
	bResetDone		: BOOL;					// Status of function block MC_Reset
	bHaltDone		: BOOL;					// Status of function block MC_Halt

	// =============== State variables ========================
	bStatusEnable	: BOOL;					// Enable feedback
	
	// =============== Velocity, override =====================
	fVelocity		: LREAL;				// Target velocity
	fOverride 		: LREAL := 100.0;		// Override 100%
	
	// =============== Trigger function blocks ================
	fbTriggerHalt	: R_TRIG;				// Trigger to recognize rising edge of halt input
	fbTriggerReset	: R_TRIG;				// Trigger to recognize rising edge of reset input
	
	// =============== Axis reference =========================
	AxisRef			: AXIS_REF;				// Axis reference (process data plc/nc)
	
	// =============== Motion function blocks =================
	fbMcPower 		: MC_Power;				// FB for enable and override
	fbMcReset 		: MC_Reset;				// FB to reset axis
	fbMcStop 		: MC_Stop;				// FB to stop axis
	fbMcHalt		: MC_Halt;				// FB to halt axis
	fbMcMove		: MC_MoveVelocity;		// FB to move axis (velocity movement)
END_VAR

// =========================================================
;
// =========================================================

PROPERTY bState_Enable : BOOL
GET
bState_Enable := bStatusEnable;
END_GET
END_PROPERTY

PROPERTY bState_HaltDone : BOOL
GET
bState_HaltDone := bHaltDone;
END_GET
END_PROPERTY

PROPERTY bState_ResetDone : BOOL
GET
bState_ResetDone := bResetDone;
END_GET
END_PROPERTY

METHOD Enable
VAR_INPUT
	bEnable		: BOOL;
END_VAR
// =========================================================

fbMCPower(	Enable 			:= bEnable, 
			Enable_Positive	:= bEnable, 
			Enable_Negative	:= bEnable, 
			Override		:= fOverride,
			Axis			:= AxisRef,
			Status			=> bStatusEnable);
			
IF fbMcPower.Error THEN
	bError		:= TRUE;
	nErrorID 	:= fbMcPower.ErrorID;
END_IF

AxisRef.ReadStatus();

bMoves := AxisRef.Status.Moving;

// =========================================================
END_METHOD

PROPERTY fTargetVelocity : LREAL
GET
fTargetVelocity := fVelocity;
END_GET
SET
fVelocity := fTargetVelocity;
END_SET
END_PROPERTY

METHOD Halt
VAR_INPUT
	bDriveHalt		: BOOL;					// Request stop
END_VAR
// =========================================================

IF bDriveHalt THEN
	// Move Execute FALSE
	fbMCMove(	Execute	:= FALSE,
				Axis 	:= AxisRef);
ELSE
	// Reset done signal
	bHaltDone := FALSE;
END_IF

// Trigger
fbTriggerHalt(CLK := bDriveHalt);

IF fbTriggerHalt.Q THEN
	fbMcHalt(	Execute	:= TRUE,
				Axis 	:= AxisRef);
ELSE
	fbMcHalt(Axis := AxisRef);
END_IF

// Done / Error / Command aborted
IF fbMcHalt.Done OR fbMcHalt.Error OR fbMcHalt.CommandAborted THEN
	bError		:= fbMcHalt.Error;
	nErrorID 	:= fbMcHalt.ErrorID;
	bHaltDone 	:= fbMcHalt.Done;
	
	fbMCMove(	Execute	:= FALSE,
				Axis 	:= AxisRef);
				
	fbMcHalt(	Execute	:= FALSE,
				Axis 	:= AxisRef);
END_IF

// =========================================================
END_METHOD

METHOD MoveBw
VAR_INPUT
END_VAR
// =========================================================

// Not error
IF NOT fbMcMove.Error THEN
	fbMCMove(	Execute 	:= TRUE,
				Velocity 	:= fVelocity,
				Direction 	:= MC_Negative_Direction,
				Axis 		:= AxisRef );
END_IF

// Error / Command aborted
IF fbMCMove.Error OR fbMCMove.CommandAborted THEN
	IF fbMcMove.Error THEN
		bError		:= TRUE;
		nErrorID 	:= fbMCMove.ErrorID;
	END_IF
	
	fbMCMove(	Execute	:= FALSE,
				Axis 	:= AxisRef);
END_IF

// =========================================================
END_METHOD

METHOD MoveFw
VAR_INPUT
END_VAR
// =========================================================

// Not error
IF NOT fbMcMove.Error THEN
	fbMCMove(	Execute 	:= TRUE,
				Velocity 	:= fVelocity,
				Direction 	:= MC_Positive_Direction,
				Axis 		:= AxisRef );
END_IF

// Error / Command aborted
IF fbMCMove.Error OR fbMCMove.CommandAborted THEN
	IF fbMcMove.Error THEN
		bError		:= TRUE;
		nErrorID 	:= fbMCMove.ErrorID;
	END_IF
	
	fbMCMove(	Execute	:= FALSE,
				Axis 	:= AxisRef);
END_IF

// =========================================================
END_METHOD

METHOD Reset
VAR_INPUT
	bDriveReset		: BOOL;					// Request reset
END_VAR
// =========================================================

IF NOT bDriveReset THEN
	bResetDone 	:= FALSE;
END_IF

// Trigger
fbTriggerReset(CLK := bDriveReset);

IF fbTriggerReset.Q THEN
	bHaltDone 	:= FALSE;
	
	fbMcReset(Execute := TRUE, Axis := AxisRef);
ELSE
	fbMcReset(Axis := AxisRef);
END_IF

// Done / Error
IF fbMcReset.Done OR fbMcReset.Error THEN
	bError		:= fbMcReset.Error;
	nErrorID 	:= fbMcReset.ErrorID;
	bResetDone 	:= fbMcReset.Done;

	fbMcReset(	Execute	:= FALSE,
				Axis 	:= AxisRef);
END_IF

// =========================================================
END_METHOD

METHOD Stop
VAR_INPUT
	bDriveStop		: BOOL;					// Request stop
END_VAR
// =========================================================

IF bDriveStop THEN
	// Move Execute FALSE
	fbMCMove(	Execute	:= FALSE,
				Axis 	:= AxisRef);
ELSE
	// Reset done signal
	bHaltDone := FALSE;
END_IF

// Trigger
fbTriggerHalt(CLK := bDriveStop);

IF fbTriggerHalt.Q THEN
	fbMcStop(	Execute	:= TRUE,
				Axis 	:= AxisRef);
ELSE
	fbMcStop(Axis := AxisRef);
END_IF

// Done / Error / Command aborted
IF fbMcStop.Done OR fbMcStop.Error OR fbMcStop.CommandAborted THEN
	bError		:= fbMcStop.Error;
	nErrorID 	:= fbMcStop.ErrorID;
	bHaltDone 	:= fbMcStop.Done;
	
	fbMCMove(	Execute	:= FALSE,
				Axis 	:= AxisRef);
				
	fbMcStop(	Execute	:= FALSE,
				Axis 	:= AxisRef);
END_IF

// =========================================================
END_METHOD

END_FUNCTION_BLOCK

// ---- 02_Subsystems/FB_Stage.TcPOU
FUNCTION_BLOCK FB_Stage
VAR_INPUT
END_VAR
VAR_OUTPUT
END_VAR
VAR
	// =============== State variables ===========================
	bHaltRequest				: BOOL;						// True if machine is in state ABORTING or STOPPING
	bResetRequest				: BOOL;						// True if machine is in state RESETTING

	// =============== Axis ======================================
	fbAxis						: FB_Axis;					// Function block instance of FB_Axis
	fAxisVelo					: LREAL;					// Velocity of axis
		
	// =============== Common variables ==========================
	fbTriggerStartingStart		: R_TRIG;					// To diagnose rising edge of starting action starting
	fbTriggerResetStart			: R_TRIG;					// To diagnose rising edge of starting reset			
	bMoved						: BOOL;						// History variable to save if axis has moved
END_VAR

END_FUNCTION_BLOCK

// ---- POUs/ModbusTCP_Test.TcPOU
PROGRAM ModbusTCP_Test
VAR
		ModBusTest : BOOL	:= 	TRUE;	//Tag_ModbusTCP<00001,OP>
END_VAR

END_PROGRAM

// ---- 05_Visu/HMI.TcVIS
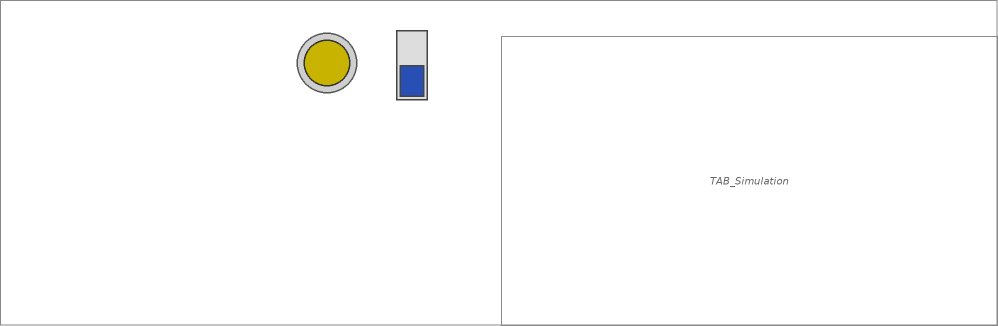
VISUALIZATION HMI  // 998x326
    TabControl (501,36 497x290)
        shows TAB_Simulation()
    DipSwitch (377,30 70x70), variable: Temp.bSwitch1, behaviour: TOGGLE, style: Switch-DipSwitch-Blue
    Lamp1 (292,28 70x70), variable: Temp.bLED1, style: Lamp-Lamp1-Yellow
END_VISUALIZATION

// ---- 05_Visu/TAB_Simulation.TcVIS
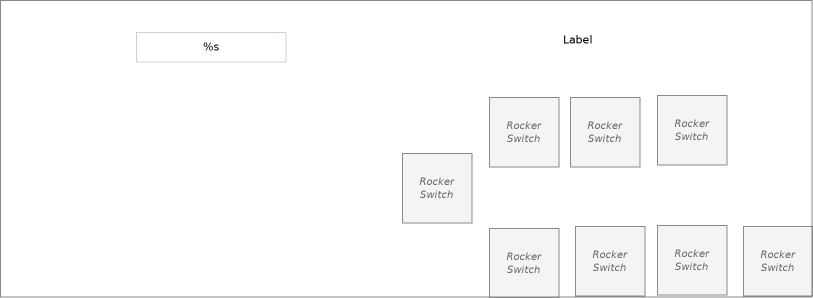
VISUALIZATION TAB_Simulation  // 813x298
    RockerSwitch (489,97 70x70), variable: MAIN.fbMachine.fbMPG.bX1, behaviour: TOGGLE, style: Switch-RockerSwitch-Blue
    RockerSwitch (570,97 70x70), variable: MAIN.fbMachine.fbMPG.bX10, behaviour: TOGGLE, style: Switch-RockerSwitch-Blue
    RockerSwitch (657,95 70x70), variable: MAIN.fbMachine.fbMPG.bX100, behaviour: TOGGLE, style: Switch-RockerSwitch-Blue
    RockerSwitch (402,153 70x70), behaviour: TOGGLE, style: Switch-RockerSwitch-Blue
    RockerSwitch (489,228 70x70), behaviour: TOGGLE, style: Switch-RockerSwitch-Blue
    RockerSwitch (575,226 70x70), behaviour: TOGGLE, style: Switch-RockerSwitch-Blue
    RockerSwitch (657,225 70x70), behaviour: TOGGLE, style: Switch-RockerSwitch-Blue
    RockerSwitch (743,226 70x70), behaviour: TOGGLE, style: Switch-RockerSwitch-Blue
    Label (503,25 150x30), "Label"
    Textfield (136,32 150x30), "%s", text variable: MAIN.fbMachine.fbVisu.sDisplayText_MPG
END_VISUALIZATION

// ---- GlobalTextList.TcGTLO
TEXTLIST GlobalTextList
  135 = '%s'
  733 = 'Label'
END_TEXTLIST
